# B&R Automation Studio project Nitto (part 11)

#### Bibliothek.fun - Exportierte Funktionen und Funktionsblöcke
```iecst
(********************************************************************
 * COPYRIGHT -- Microsoft
 ********************************************************************
 * Library: Bibliothek
 * Datei: Bibliothek.fun
 * Autor: Awalz
 * Erstellt: 31. März 2014
 ********************************************************************
 * Funktionen und Funktionsblöcke der Library Bibliothek
 ********************************************************************)

FUNCTION_BLOCK FB_CONST_MACHINE_MODES (*TODO: Bitte Kommentar hier einzufügen*)
	VAR_OUTPUT
		MANUAL : INT := 0;
		AUTOMATIC : INT := 1;
		PRODUCTION : INT := 2;
		SAFETYSTOP : INT := 7;
		RESET : INT := 8;
		EMERGENCYSTOP : INT := 9; (*texts : ARRAY[MANUAL..EMERGENCYSTOP] OF STRING[20] := ['MANUAL','AUTOMATIC','PRODUCTION','***3***','***4***','***5***','***6***','SAFETYSTOP','RESET','EMERGENCYSTOP'];*)
		texts : ARRAY[0..9] OF STRING[20] := ['MANUAL','AUTOMATIC','PRODUCTION','***3***','***4***','***5***','***6***','SAFETYSTOP','RESET','EMERGENCYSTOP'];
	END_VAR
END_FUNCTION_BLOCK

FUNCTION_BLOCK FB_CONST_AXIS_ACTIONS (*TODO: Bitte Kommentar hier einzufügen*)
	VAR_OUTPUT
		NOACTION : INT := 0;
		START : INT := 1;
		CALIBR : INT := 2;
		JOG_POS : INT := 3;
		JOG_NEG : INT := 4;
		SETPOS : INT := 6;
		CPLON : INT := 7;
		CPLOFF : INT := 8;
		STOP : INT := 9;
		RESET : INT := 10;
		OPEN : INT := 11; (* Break Open*)
		CLOSE : INT := 12; (* Break Close*)
		WRITE : INT := 13; (* Write Parameter*)
		READ : INT := 14; (* Read Parameter*)
		MOVE_VELOCITY : INT := 15;
		POWER_ON : INT := 16;
		VAXIS_ON : INT := 17;
		POWER_OFF : INT := 18;
		MOVE_CYCLIC_VELOCITY : INT := 20;
		SETPOSREL : INT := 21;
		SETPOSREL_NOLIMIT : INT := 22;
		EMERGENCY_DECELERATION : REAL := 1111111; (*200m/min 200*16666.67/2 in 2 sek*)
		texts : ARRAY[0..19] OF STRING[15] := ['NOACTION','START','CALIBR','JOG_POS','JOG_NEG','SETPOS','SETPOS','CPLON','CPLOFF','STOP','RESET','OPEN','CLOSE','WRITE','READ','MOVE_VELO','POWER_ON','VAXIS_ON','POWER_OFF'];
	END_VAR
END_FUNCTION_BLOCK

FUNCTION_BLOCK FB_CONST_MASCHINE (*TODO: Bitte Kommentar hier einzufügen*)
	VAR_INPUT
		MACHINEMODES : FB_CONST_MACHINE_MODES;
		AXIS : FB_CONST_AXIS_ACTIONS;
		LAMP : FB_CONST_LAMP;
		CUTTINGUNIT : FB_CONST_CUTTINGUNIT;
		UNITMODEs : FB_CONST_UNIT_MODES;
		ALARMS : FB_CONST_ALARMS;
	END_VAR
END_FUNCTION_BLOCK

FUNCTION_BLOCK FB_ClkPulse (*TODO: Bitte Kommentar hier einzufügen*)
	VAR_INPUT
		enable : BOOL;
		TimeOn : TIME := T#100ms;
		TimeOff : TIME := T#100ms;
	END_VAR
	VAR_OUTPUT
		Output : BOOL := FALSE;
	END_VAR
	VAR CONSTANT
		CLOCK_ON : INT := 0;
		CLOCK_WAIT_ON : INT := 1;
		CLOCK_WAIT_OFF : INT := 3;
	END_VAR
	VAR
		state : INT := CLOCK_ON;
		timer : TON;
	END_VAR
END_FUNCTION_BLOCK

FUNCTION_BLOCK FB_Clk (*TODO: Bitte Kommentar hier einzufügen*)
	VAR_OUTPUT
		c500 : FB_ClkPulse := (enable:=TRUE,TimeOn:=T#500ms,TimeOff:=T#500ms);
		c200 : FB_ClkPulse := (enable:=TRUE,TimeOn:=T#200ms,TimeOff:=T#200ms);
		c1000 : FB_ClkPulse := (enable:=TRUE,TimeOn:=T#1000ms,TimeOff:=T#1000ms);
		c5000 : FB_ClkPulse := (enable:=TRUE,TimeOn:=T#5000ms,TimeOff:=T#5000ms);
	END_VAR
END_FUNCTION_BLOCK

FUNCTION_BLOCK FB_CONST_LAMP (*TODO: Bitte Kommentar hier einzufügen*)
	VAR_OUTPUT
		OFF : INT := 0;
		ON : INT := 1;
		BLINK200 : INT := 2;
		BLINK500 : INT := 3;
		BLINK1000 : INT := 4;
		BLINK5000 : INT := 5;
	END_VAR
END_FUNCTION_BLOCK

FUNCTION_BLOCK FB_CONST_CUTTINGUNIT (*TODO: Bitte Kommentar hier einzufügen*)
	VAR_INPUT
		MODEs : FB_CONST_CUTTINGUNIT_MODES;
		CMDs : FB_CONST_CUTTINGUNIT_CMDS;
		ERRORs : FB_CONST_CUTTINGUNIT_ERRORS;
		TOOLs : FB_CONST_CUTTINGUNIT_TOOLS;
	END_VAR
END_FUNCTION_BLOCK

FUNCTION_BLOCK FB_CONST_CUTTINGUNIT_MODES (*TODO: Bitte Kommentar hier einzufügen*)
	VAR_OUTPUT
		DISABLE : UDINT := 0; (*BYTE *) (* nicht gekoppelt zur Achse vom Mastermodul *)
		FREE_RUN : UDINT := 1; (*BYTE *) (* freies Schneiden *)
		SYNC_RUN : UDINT := 2; (*BYTE *) (* synchronisieren z.B. Registermarken *)
		CROSS_CUT : UDINT := 3;
		END_MODE : UDINT := 10; (*BYTE *)
		texts : ARRAY[1..4] OF STRING[20] := ['DISABLE','FREE_RUN','SYNC_RUN','CROSS_CUT'];
	END_VAR
END_FUNCTION_BLOCK

FUNCTION_BLOCK FB_CONST_CUTTINGUNIT_CMDS (*TODO: Bitte Kommentar hier einzufügen*)
	VAR_OUTPUT
		NO_CMD : INT := 0;
		CALIBR : INT := 1;
		INIT : INT := 2;
		CPL_ON : INT := 3;
		CPL_OFF : INT := 4;
		DEINIT : INT := 5;
		SYNC : INT := 6;
		MOVEFW : INT := 7;
		MOVEBW : INT := 8;
		RESET : INT := 9;
		SETDATA : INT := 10;
		ABORT : INT := 11;
		texts : ARRAY[1..11] OF STRING[20] := ['NO_CMD','CALIBR','INT','CPL_ON','CPL_OFF','DEINIT','SYNC','MOVEFW','MOVEBW','RESET','SETDATA','ABORT'];
	END_VAR
END_FUNCTION_BLOCK

FUNCTION_BLOCK FB_CONST_UNIT_MODES (*TODO: Bitte Kommentar hier einzufügen*)
	VAR_OUTPUT
		DISABLE : UDINT := 0; (*BYTE*)
		ENABLE : UDINT := 1; (*BYTE*)
		AXIS_OFF : DINT := 2;
		texts : ARRAY[0..2] OF STRING[20] := ['DISABLE','ENABLE','AXIS_OFF'];
	END_VAR
END_FUNCTION_BLOCK

FUNCTION_BLOCK FB_CUTTINGUNIT_CMD (*TODO: Bitte Kommentar hier einzufügen*)
	VAR_INPUT
		value : INT;
		set : BOOL;
	END_VAR
	VAR_OUTPUT
		text : STRING[20];
	END_VAR
	VAR
		CONST : FB_CONST_MASCHINE;
	END_VAR
END_FUNCTION_BLOCK

FUNCTION_BLOCK FB_TensionMeasure (*TODO: Bitte Kommentar hier einzufügen*)
	VAR_INPUT
		offsetVisu : LREAL;
		data : FB_TENSIONMEASUREDATA;
		init : BOOL;
	END_VAR
	VAR_OUTPUT
		status : FB_ModulStatus;
		actValue : LREAL;
	END_VAR
	VAR
		CyclicWrite : MC_BR_CyclicWrite;
		PIDControler : LCRPID; (* PID REGLER*)
		LCRPIDpara_TM : LCRPIDpara; (* Parameter für PID REGLER*)
		FilterPT1 : LCRPT1e;
		CONST : FB_CONST_MASCHINE;
	END_VAR
	VAR CONSTANT
		STEP_TM_INIT1 : USINT := 0; (*Initialisation step 1*)
		TENSION_T_FILTER : REAL := 0.016; (*tension filter time [s]*)
		STEP_TM_WAIT_POWER_ENABLED : USINT := 7; (*Wait until all available axes are enabled*)
		STEP_TM_READY : USINT := 10; (*General state after initialisation, waining for commands*)
		STEP_TM_LOAD_PARA_START : USINT := 20; (*Start parameter loading (e.g. PID controller parameter)*)
		STEP_TM_WAIT_LOAD_PARA_DONE : USINT := 21; (*Wait for parameter being loaded *)
		STEP_TM_WAIT_SWITCH_CTRL_ON : USINT := 40; (*Switch PID controller on*)
		STEP_TM_CTRL_ACTIVE : USINT := 41; (*Wait for commands in active control*)
		STEP_TM_CTRL_PAUSE : USINT := 42; (*Pausing control until the master velocity is back in the required range*)
		STEP_TM_CTRL_OFF : USINT := 43; (*Switch off web tension control*)
	END_VAR
END_FUNCTION_BLOCK

FUNCTION_BLOCK FB_TENSIONMEASUREDATA (*TODO: Bitte Kommentar hier einzufügen*)
	VAR_INPUT
		mode : UDINT; (*BYTE;*)
		setvalue : REAL;
	END_VAR
	VAR_OUTPUT
		newRecipe : BOOL;
	END_VAR
END_FUNCTION_BLOCK

FUNCTION_BLOCK FB_Safety (*TODO: Bitte Kommentar hier einzufügen*)
	VAR_INPUT
		ResetSafeMC : BOOL; (*Reset input of SafeMC Function Blocks*)
		ResetStartupInhibit : BOOL; (*Reset emergency functions (quit startup inhibit)*)
		ResetUserSafeMC : BOOL;
		SLSmasterVeloScaled : REAL;
		Control_OFF : BOOL;
		CtrlPowerEmcyDel : BOOL;
		CtrlPowerEmcyUndel : BOOL; (* schaltet die Schützte für 24V Versorgung*)
		EnabDrives : BOOL;
		manuelmode : BOOL;
	END_VAR
	VAR_OUTPUT
		RequestSTO : BOOL; (*Emergency Stop is requested (active low)*)
		RequestSLS : BOOL; (*Safe Limited Speed requested by opening safety doors (active low)*)
		Request_ONdelay : BOOL;
		valid : BOOL;
	END_VAR
END_FUNCTION_BLOCK

FUNCTION_BLOCK FB_ModulStatus (*TODO: Bitte Kommentar hier einzufügen*)
	VAR_INPUT
		id : UINT;
		name : STRING[30];
		isCoupled : BOOL;
		mode : UDINT; (* BYTE;*)
		ready : BOOL;
		reverse : BOOL;
		axiserror : BOOL;
	END_VAR
	VAR_OUTPUT
		modeName : STRING[80];
		error : BOOL;
		AxisState_status : STRING[20];
	END_VAR
	VAR_IN_OUT
		axisState : MC_ReadStatus;
	END_VAR
END_FUNCTION_BLOCK

FUNCTION_BLOCK FB_Ampel (*TODO: Bitte Kommentar hier einzufügen*)
	VAR_INPUT
		Rot : FB_Lamp; (*DiDo_Type;*)
		Gelb : FB_Lamp; (*DiDo_Type;*)
		Gruen : FB_Lamp; (* DiDo_Type;*)
		horn : BOOL;
		hornoff : BOOL;
		hornPuls : FB_Lamp;
		ondelay : TIME;
	END_VAR
	VAR_OUTPUT
		horn_o : BOOL;
	END_VAR
	VAR_IN_OUT
		clk : FB_Clk;
	END_VAR
	VAR
		rtrig : R_TRIG;
		timer_TOF : TOF;
		timer_TON : TON;
	END_VAR
END_FUNCTION_BLOCK

FUNCTION_BLOCK FB_Lamp (*TODO: Bitte Kommentar hier einzufügen*)
	VAR_INPUT
		aktion : INT := 0;
	END_VAR
	VAR_OUTPUT
		led : BOOL := FALSE;
		ledinv : BOOL := FALSE;
		button : BOOL;
		rtrig : R_TRIG;
		ftrig : F_TRIG;
	END_VAR
	VAR_IN_OUT
		clk : FB_Clk;
	END_VAR
	VAR
		CONST : FB_CONST_MASCHINE;
		output : BOOL := FALSE;
	END_VAR
END_FUNCTION_BLOCK

FUNCTION_BLOCK FB_KeyLamp (*TODO: Bitte Kommentar hier einzufügen*)
	VAR_INPUT
		LDT : FB_Lamp;
	END_VAR
	VAR_IN_OUT
		clk : FB_Clk;
	END_VAR
END_FUNCTION_BLOCK

FUNCTION_BLOCK FB_UnitChkStatus (*TODO: Bitte Kommentar hier einzufügen*)
	VAR_INPUT
		enable : BOOL;
		setMode : UDINT; (*BYTE;*)
	END_VAR
	VAR_OUTPUT
		ready : BOOL;
	END_VAR
	VAR_IN_OUT
		status : FB_ModulStatus;
	END_VAR
	VAR
		CONST : FB_CONST_MASCHINE;
	END_VAR
END_FUNCTION_BLOCK

FUNCTION_BLOCK FB_PullBreakClampToggle (*TODO: Bitte Kommentar hier einzufügen*)
	VAR_INPUT
		buttomToggle : FB_KeyLamp;
		buttomToggle2 : FB_KeyLamp;
		limiterSwitchDrvSide : BOOL;
		limiterSwitchOpSide : BOOL;
		isup : BOOL;
		isdown : BOOL;
		enable : BOOL;
		init : BOOL;
		onewayini : BOOL;
	END_VAR
	VAR_OUTPUT
		toUp_o : BOOL;
		toDown_o : BOOL;
		limiterBackward_o : BOOL;
		limiterForward_o : BOOL;
	END_VAR
	VAR_IN_OUT
		clk : FB_Clk;
	END_VAR
	VAR
		Time1 : TON;
		state : USINT := 0;
		CONST : FB_CONST_MASCHINE;
	END_VAR
END_FUNCTION_BLOCK

FUNCTION_BLOCK FB_ErrorHdl (*TODO: Bitte Kommentar hier einzufügen*)
	VAR_INPUT
		set : BOOL;
		reset : BOOL;
		flag : BOOL;
		id : DINT;
		state : DINT;
		text : STRING[256];
		fnc : STRING[128];
	END_VAR
END_FUNCTION_BLOCK

FUNCTION_BLOCK FB_Panel (*TODO: Bitte Kommentar hier einzufügen*)
	VAR_INPUT
		Emergency : FB_KeyLamp;
		EMCY_Button : BOOL;
		LDTRESET : FB_KeyLamp;
		LDTStop : FB_KeyLamp;
		LDTAutomatic : FB_KeyLamp;
		LDTJOG : FB_KeyLamp;
		LDTControlON : FB_KeyLamp;
		LDTControlOFF : FB_KeyLamp;
	END_VAR
	VAR_OUTPUT
		clk : FB_Clk;
		EMCY_Button_o : INT;
	END_VAR
END_FUNCTION_BLOCK

FUNCTION_BLOCK FB_CONVEYOR_DATA (*TODO: Bitte Kommentar hier einzufügen*)
	VAR_INPUT
		gap : LREAL;
		pcs : INT;
		newParam2 : BOOL;
	END_VAR
END_FUNCTION_BLOCK

FUNCTION_BLOCK FB_MASTERMODUL_DATA (*TODO: Bitte Kommentar hier einzufügen*)
	VAR_INPUT
		speedToCycleWebturrit : REAL;
		startSpeed : REAL;
		maxSpeed : REAL;
		periodLength : REAL;
		lenght1 : REAL;
		lenght2 : REAL;
	END_VAR
END_FUNCTION_BLOCK

FUNCTION_BLOCK FB_MessageInstance (*TODO: Bitte Kommentar hier einzufügen*)
	VAR_INPUT
		active : BOOL;
		InstanceId : UDINT; (* Aggregat, Instaziertes Objekt *)
		ErrorId : UDINT;
		StationName : STRING[20];
	END_VAR
	VAR_OUTPUT
		err : FB_ErrorHdl;
		busy : BOOL;
	END_VAR
	VAR
		state : INT;
		sFormatString : STRING[29] := '';
		arrParaPointer : ARRAY[1..3] OF DINT;
		sPara1 : STRING[20];
		nPara2 : DINT;
		nPara3 : DINT; (*fbLogEvent:		ADSLOGEVENT := ( PORT:=110,
											  TMOUT := T#2s,
											  EventConfigData := ( 	Class := TCEVENTCLASS_ALARM,
																			Prio := TCEVENTPRIO_IMPLICIT,
																			ProgId := 'TcEventFormatter.TcXmlFormatter',
																			StreamType := TCEVENTSTREAM_NORMAL,
																			bQuitRequired := FALSE
																		)
											);*)
	END_VAR
END_FUNCTION_BLOCK

FUNCTION_BLOCK FB_WinderData (*TODO: Bitte Kommentar hier einzufügen*)
	VAR_INPUT
		recipeData : FB_WinderRecipeData;
		machData : FB_WinderMachData;
	END_VAR
END_FUNCTION_BLOCK

FUNCTION_BLOCK FB_WinderRecipeData (*TODO: Bitte Kommentar hier einzufügen*)
	VAR_INPUT
		stopDiam : UDINT;
		warnDiam : UDINT;
		minDiamTension : UDINT; (*Mode*)
		maxDiamTension : UDINT; (*Mode*)
		mode : UDINT; (*Mode*)
		reverse : BOOL;
		dancersolPos : REAL;
	END_VAR
END_FUNCTION_BLOCK

FUNCTION_BLOCK FB_WinderMachData (*TODO: Bitte Kommentar hier einzufügen*)
	VAR_INPUT
		coreDiam : UDINT;
		frictionCompensation : USINT := 0;
		velocityOverride : USINT := 0;
		GEAR_RATIO : REAL;
		axistyp : SINT; (* (-1: winder, +1: unwinder).*)
	END_VAR
END_FUNCTION_BLOCK

FUNCTION_BLOCK FB_ScalingPerimeter (*TODO: Bitte Kommentar hier einzufügen*)
	VAR_INPUT
		realperimeter : REAL; (* Umfang des Wekrzeuges *)
		NumberToolSegments : USINT; (*Anzahl der Nutzen auf dem Werkzeug/Stanzblech*)
	END_VAR
	VAR_OUTPUT
		Scaledperimeter : UDINT;
		ToolSegmentPeriod : UDINT;
	END_VAR
	VAR
		Remainder : DINT;
	END_VAR
END_FUNCTION_BLOCK

FUNCTION_BLOCK FB_CUTTINGUNIT_STATUS (*TODO: Bitte Kommentar hier einzufügen*)
	VAR_INPUT
		id : UINT;
		tableid : UINT;
		name : STRING[30];
		dataOk : BOOL;
		isCalibrated : BOOL;
		isInitialized : BOOL;
		isCoupled : BOOL;
		isSynchronized : BOOL; (*	errors:					FB_CUTTINGUNIT_ERRORS;*) (*tmpData:				FB_CUTTINGUNIT_TMPDATA;*)
		errorstop : BOOL;
		extReady : BOOL := TRUE;
		mode : FB_CUTTING_MODE;
	END_VAR
	VAR_OUTPUT
		ready : BOOL;
		tmpCalibrated : BOOL;
		AxisState_status : STRING[20];
	END_VAR
	VAR_IN_OUT
		recipeMode : UDINT; (*	BYTE;*)
		axisState : MC_ReadStatus;
	END_VAR
	VAR
		CONST : FB_CONST_MASCHINE;
	END_VAR
END_FUNCTION_BLOCK

FUNCTION_BLOCK FB_CUTTING_MODE (*TODO: Bitte Kommentar hier einzufügen*)
	VAR_INPUT
		value : UDINT; (*BYTE;*)
	END_VAR
	VAR_OUTPUT
		text : STRING[20];
	END_VAR
	VAR
		CONST : FB_CONST_MASCHINE;
	END_VAR
END_FUNCTION_BLOCK

FUNCTION_BLOCK FB_PowerBridge (*TODO: Bitte Kommentar hier einzufügen*)
	VAR_INPUT
		bridgedownbutton : FB_CLAMP;
		withpressureSensor : BOOL;
		movebutton : FB_KeyLamp;
	END_VAR
	VAR_OUTPUT
		pressuredrvside : INT;
		pressureOperside : INT;
		button : BOOL; (*Button in der Visu*)
		valveOut : BOOL;
		pressurepresent : BOOL;
		toggle : FB_PullBreakClampToggle;
	END_VAR
	VAR_IN_OUT
		clk : FB_Clk;
	END_VAR
	VAR
		KNpressuredrvside : REAL;
		KNpressureOperside : REAL;
		pressurereference : REAL;
	END_VAR
	VAR CONSTANT
		SCALE_10V_TO_KN : REAL := (10.0/32767.0); (*10.0 V = 10 kN; 10.0 V = 32767*)
	END_VAR
END_FUNCTION_BLOCK

FUNCTION_BLOCK FB_CONST_CUTTINGUNIT_ERRORS (*TODO: Bitte Kommentar hier einzufügen*)
	VAR_OUTPUT
		REF_ERROR_UNIT_CLOSED : INT := 1;
		AXISERROR : INT := 2;
		SAFETY_SPEED : INT := 3;
		HAUBE1_VORN_OFFEN : INT := 8;
		HAUBE2_HINTEN_OFFEN : INT := 9;
		RECIPE_MODE_UNDEF : INT := 30;
		RECIPE_TOOLNR : INT := 31;
		RECIPE_SHAPE_CONFIG : INT := 32;
		CUTTER_DIAMETER : INT := 33;
		CUTTER_ZAEHNE : INT := 34;
		ANVILROLLER_ZAEHNE : INT := 35;
		ERROR_TABLE_CALC : INT := 36;
	END_VAR
END_FUNCTION_BLOCK

FUNCTION_BLOCK FB_CONST_CUTTINGUNIT_TOOLS (*TODO: Bitte Kommentar hier einzufügen*)
	VAR_OUTPUT
		MIN_TOOLS : INT := 1;
		MAX_TOOLS : INT := 1000;
	END_VAR
END_FUNCTION_BLOCK

FUNCTION_BLOCK FB_TurnGrWinKeysbox (*TODO: Bitte Kommentar hier einzufügen*)
	VAR_INPUT
		GridWinrightkey : FB_CLAMP;
		GridWinleftkey : FB_CLAMP;
		feederturnkey : FB_KeyLamp;
	END_VAR
	VAR_OUTPUT
		feederlimitswitch : BOOL;
		feederturn : BOOL;
		feederright : BOOL;
	END_VAR
	VAR_IN_OUT
		clk : FB_Clk;
	END_VAR
END_FUNCTION_BLOCK

FUNCTION_BLOCK FB_SPLICETABLE (*TODO: Bitte Kommentar hier einzufügen*)
	VAR_INPUT
		disable : BOOL;
		clampBefore : FB_CLAMP;
		clampAfter : FB_CLAMP;
	END_VAR
	VAR_OUTPUT
		ready : BOOL;
	END_VAR
	VAR_IN_OUT
		clk : FB_Clk;
	END_VAR
END_FUNCTION_BLOCK

FUNCTION_BLOCK FB_CLAMP (*TODO: Bitte Kommentar hier einzufügen*)
	VAR_INPUT
		buttonDown : FB_KeyLamp;
		buttonvisu : BOOL;
		toDown_o : BOOL;
		disable : BOOL;
	END_VAR
	VAR_IN_OUT
		clk : FB_Clk;
	END_VAR
	VAR
		visutrigg : R_TRIG;
		CONST : FB_CONST_MASCHINE;
	END_VAR
END_FUNCTION_BLOCK

FUNCTION_BLOCK FB_Cylinder (*TODO: Bitte Kommentar hier einzufügen*)
	VAR_INPUT
		upVISU : BOOL;
		downVISU : BOOL;
		buttonUP : BOOL;
		buttonDown : BOOL;
		Enable : BOOL;
		up_o : BOOL;
		down_o : BOOL;
	END_VAR
	VAR_OUTPUT
		isUp : BOOL;
		isDown : BOOL;
		isdowndelayed : BOOL;
	END_VAR
	VAR
		timer : TON;
	END_VAR
END_FUNCTION_BLOCK

FUNCTION_BLOCK FB_Hydraulic (*TODO: Bitte Kommentar hier einfügen*) (*$GROUP=Anwender*)
	VAR_INPUT
		enable : BOOL;
		buttonDown : BOOL;
		buttonUp : BOOL;
		limitswitch : BOOL; (* kein Endschalter für untern da nur Ventile aufgemacht werden und der Wickler drucklos bis zum Ende fährt*)
	END_VAR
	VAR_OUTPUT
		go_up : BOOL; (*go_down:		BOOL;*) (* da kein Ventil angesteuert wird nur das Ventil für hoch gelüftet wird*)
		commonValve : BOOL;
		LED_is_up : BOOL;
		LED_is_down : BOOL;
		pumpe : BOOL;
	END_VAR
END_FUNCTION_BLOCK

FUNCTION_BLOCK FB_UnwinderfeederCtrl (*TODO: Bitte Kommentar hier einfügen*) (*$GROUP=Anwender*)
	VAR_INPUT
		cmd : INT;
		buttonRequestOpSide : FB_KeyLamp;
		buttonRightOpSide : FB_KeyLamp;
		buttonLeftOpSide : FB_KeyLamp;
		buttonRequestDrvSide : FB_KeyLamp;
		buttonRightDrvSide : FB_KeyLamp;
		buttonLeftDrvSide : FB_KeyLamp;
		LimitSwitchRight : BOOL;
		LimitSwitchLeft : BOOL;
		axisREF : UDINT;
		UnwFeeder_HW : SdcHwCfg_typ := (0);
		UnwFeeder_DrvIf : SdcDrvIf16_typ := (0);
		UnwFeeder_DiDoIf : SdcDiDoIf_typ := (0);
		UnwFeeder_ModuleOk : BOOL := 0;
		UnwFeederErrorAckn : BOOL;
		BasicControl : basic_typ;
	END_VAR
	VAR_OUTPUT
		feederFUleft : BOOL;
		feederFUright : BOOL;
		brakerelease : BOOL;
		ampelgelb : BOOL;
		horn : BOOL;
		MC_ReadStatus_0 : MC_ReadStatus;
		busy : BOOL;
		status : FB_ModulStatus;
	END_VAR
	VAR_IN_OUT
		machineaxis : FB_AxisCtrl;
		clk : FB_Clk;
	END_VAR
	VAR
		AxisStep : INT;
		cmdtmp : INT;
		trigOPSide : BOOL;
		trigDrvSide : BOOL;
		braketimer : BOOL;
		MC_BR_ReadDriveStatus_0 : MC_BR_ReadDriveStatus;
		firststart : BOOL := TRUE;
		State : USINT;
		CONST : FB_CONST_MASCHINE;
		MC_BR_JogVelocity_0 : MC_BR_JogVelocity;
		pAxis : REFERENCE TO ACP10AXIS_typ;
		MC_Power_0 : MC_Power;
		MC_Stop_0 : MC_Stop;
		MC_Reset_0 : MC_Reset;
		Start_timer : BOOL; (*timer_TOF : TON;*)
		timer_TON : TON;
		timerOPside_TOF : TOF; (*Scahltet den Regler ab und damit fällt die Bremse zu*)
		timerDrvside_TOF : TOF;
		timer_TP : TP;
	END_VAR
	VAR CONSTANT
		STATE_READY : INT := 0;
		STATE_POWER_ON : INT := 10;
		STATE_POWER_OFF : INT := 11;
		STATE_ERROR_RESET : INT := 12;
		STATE_QUIT : INT := 20;
		ST_WAIT : USINT := 0;
		ST_REQUEST : USINT := 10;
		ST_REQUEST_OpSide : USINT := 20;
		ST_REQUEST_DrvSide : USINT := 30;
		ST_END : USINT := 40;
	END_VAR
END_FUNCTION_BLOCK

FUNCTION_BLOCK FB_DUBBLEUUNWINDERDATA (*TODO: Bitte Kommentar hier einfügen*) (*$GROUP=Anwender*)
	VAR_INPUT
		undwinderDRV : FB_WinderData; (*drive side*)
		unwinderOP : FB_WinderData; (*operator side*)
	END_VAR
END_FUNCTION_BLOCK

FUNCTION_BLOCK FB_UNWINDERUNITSTATUS (*TODO: Bitte Kommentar hier einfügen*) (*$GROUP=Anwender*)
	VAR_INPUT
		statusDrv : FB_ModulStatus;
		statusOP : FB_ModulStatus;
	END_VAR
END_FUNCTION_BLOCK

FUNCTION_BLOCK FB_limitswitch (*TODO: Bitte Kommentar hier einfügen*) (*$GROUP=Anwender*)
	VAR_INPUT
		limitSWupper : BOOL;
		limitSWlower : BOOL;
		mechbrake : BOOL;
	END_VAR
END_FUNCTION_BLOCK

FUNCTION_BLOCK FB_StartStopbox (*TODO: Bitte Kommentar hier einfügen*) (*$GROUP=Anwender*)
	VAR_INPUT
		start : FB_KeyLamp;
		stop : FB_KeyLamp;
		jog : FB_KeyLamp;
	END_VAR
	VAR_IN_OUT
		clk : FB_Clk;
	END_VAR
END_FUNCTION_BLOCK

FUNCTION_BLOCK FB_SummeryStarStop (*TODO: Bitte Kommentar hier einfügen*) (*$GROUP=Anwender*)
	VAR_INPUT
		boxunwinder : FB_StartStopbox;
		boxwebbuffer : FB_StartStopbox;
		boxcutting1 : FB_StartStopbox;
		boxlongcutter : FB_StartStopbox;
		boxconveyor : FB_StartStopbox;
	END_VAR
	VAR_OUTPUT
		start : BOOL;
		stop : BOOL;
		jog : BOOL;
	END_VAR
	VAR_IN_OUT
		panel : FB_Panel;
		clk : FB_Clk;
	END_VAR
END_FUNCTION_BLOCK

FUNCTION_BLOCK FB_WebGuiding (*TODO: Bitte Kommentar hier einfügen*) (*$GROUP=Anwender*)
	VAR_INPUT
		enable : BOOL;
		center : BOOL;
		auto : BOOL;
		hand : BOOL;
		moveRight : BOOL;
		moveLeft : BOOL;
		hardwareOK : BOOL;
	END_VAR
	VAR_OUTPUT
		manual : BOOL;
		neutral : BOOL;
		automatic : BOOL;
		centerSelect : BOOL;
		handSelect : BOOL;
		autoSelect : BOOL;
		active : BOOL;
		arrowRight : BOOL;
		arrowLeft : BOOL;
		hardwareActive : BOOL;
	END_VAR
	VAR
		TP_01 : TP;
		Start_timer : BOOL;
		handtrigg : R_TRIG;
		centertrigg : R_TRIG;
		autotrigg : R_TRIG;
	END_VAR
END_FUNCTION_BLOCK

FUNCTION_BLOCK FB_SetGearRatio (*TODO: Bitte Kommentar hier einfügen*) (*$GROUP=Anwender*)
	VAR_INPUT
		UpdateRecipe : BOOL;
		setvalueVisuRecipe : REAL;
		enable : BOOL;
		step1 : BOOL;
		step10 : BOOL;
		step100 : BOOL;
		gearup : BOOL;
		gearlow : BOOL;
		Selectstep1 : BOOL;
		Selectstep10 : BOOL;
		Selectstep100 : BOOL;
		Selectenable : BOOL;
		limitvisupos : REAL;
		limitvisuneg : REAL;
		limitratiopos : INT;
		limitrationeg : INT;
		init : BOOL;
	END_VAR
	VAR_OUTPUT
		trigger : BOOL;
		ratioNumeratorOut : INT;
		ratioDenominator : UINT := 1000;
		setvalueVisu : REAL;
		stepvisu : REAL;
		ratio_inProcent_visu : REAL;
	END_VAR
	VAR
		offsetrecipe : REAL;
		trigP : R_TRIG;
		trigN : R_TRIG;
		ratio : INT := 1000;
		ratiotmp : INT;
		step : INT;
		TP_01 : TP;
		Start_timer : BOOL;
	END_VAR
END_FUNCTION_BLOCK

FUNCTION_BLOCK FB_MarkPoints (*TODO: Bitte Kommentar hier einfügen*) (*$GROUP=Anwender*)
	VAR_INPUT
		MC_BR_TouchProbe_0 : MC_BR_TouchProbe;
		reset : BOOL;
		Enable : BOOL;
		TriggerInput : MC_BR_TRIGGER_REF; (*Input that is used as event source*)
		Axis : UDINT; (*Axis reference of slave*)
		SearchRM : BOOL; (*Initiate search of new RM on positive edge*)
		CutMasterPosition : DINT; (*Uncorrected next cut position [Master Units]*)
		RegMarkPosition : DINT; (*RegMark offset relative to cut position [Master Units]*)
		WindowNegative : REAL; (*Range before the expected position in which the trigger signal may occur [Master Units]*)
		WindowPositive : REAL; (*Range after the expected position in which the trigger signal may occur [Master Units]*)
		ProductLength : REAL; (*Interval between two expected trigger positions [Master Units]*)
		markpointlist : FB_Markpointarray;
	END_VAR
	VAR_OUTPUT
		RecordedValue : DINT; (*Most recent RM position [Master Units]*)
		lastrecocordedValue : DINT; (*last Position befor RM lost [Master Units]*)
		ProbeCounter : UDINT; (*Number of valid trigger events. Reset by "SearchRM"*)
		MissedTriggers : UDINT; (*Number of invalid or missed trigger events. Reset by "SearchRM"*)
		CorrectionValue : DINT; (*Deviation between corrected and uncorrected cut position [Master Units]. Can be used as a relative distance for correction movements.*)
		CorrectionValid : BOOL; (*TRUE for 1 cycle if "CorrectionValue" is valid. Can be used to trigger correction movements.*)
		ActProductLength : REAL; (*Actual measured product length*)
		Active : BOOL; (*FB is enabled - waiting for a trigger event*)
		Busy : BOOL; (*FB is not yet finished*)
		Error : BOOL; (*Error occurred in FB*)
		ErrorID : UINT; (*Error number*)
	END_VAR
END_FUNCTION_BLOCK

FUNCTION_BLOCK FB_CROSSCUTPAR (*TODO: Bitte Kommentar hier einfügen*) (*$GROUP=Anwender*)
	VAR_INPUT
		StartMasterVelocity : REAL; (*Master velocity at very first cut [Master Units/ s]*)
		MaxMasterVelocity : REAL; (*Maximum master velocity [Master Units/ s]*)
		Insetting : REAL; (*Insetting ratio for calculation of CutRangeMaster [%]*)
		MaxCorrection : DINT; (*Maximum correction movement per product cycle [Master Units]*)
		CutStartPos : DINT; (*Start of synchronisation within slave period [Slave Units]*)
		CutEndPos : DINT; (*End of synchronisation within slave period [Slave Units]*)
		CutRangeMaster : REAL;
		CutRangeSlave : REAL;
		ProductLength : REAL;
		CutPosition : REAL;
		StartMode : UINT;
		ProductLengthCorrection : REAL;
		MasterStartDistance : REAL;
		StartInterval : REAL;
		MinCutRangeSlave : REAL; (*Minimum synchronization distance [Slave Units]*)
		MinCompRangeSlave : REAL; (*Minimum effective compensation distance [Slave Units]*)
	END_VAR
END_FUNCTION_BLOCK

FUNCTION_BLOCK FB_GetNextCuttPos (*TODO: Bitte Kommentar hier einfügen*) (*$GROUP=Anwender*)
	VAR_INPUT
		Enable : BOOL;
		reset : BOOL;
		donecut : BOOL; (*wait until Cutter is done with a cut*)
		RecordedValue : DINT; (*Recorded RegMark position, e.g. from a MC_BR_Touchprobe instance [Master Units]*)
		RecordedValueValid : BOOL;
		CutPosition : DINT; (*Uncorrected next cut position [Master Units]*)
		DistanceToSensor : DINT; (*Distance between tool and sensor [Master Units]*)
		RegMarkPosition : DINT; (*RegMark offset relative to cut position [Master Units]*)
		ProductLength : DINT; (*Product length [Master Units]*) (*	Touchpobe: MC_BR_TouchProbe;*)
		setCutOffset : FB_SetCutOffset;
	END_VAR
	VAR_OUTPUT
		PositionError : DINT; (*Difference between corrected and uncorrected cut position [Master Units]*)
		PositionErrorValid : BOOL; (*TRUE for 1 cycle if "PositionError" is within current product cycle*)
		nextsyncpos : DINT; (* Position für die Sunchronisierung der Stanze /Querschneider*)
		newdata : UDINT;
	END_VAR
	VAR_IN_OUT
		markpoints : FB_MarkPoints;
		scalePerimeter : FB_ScalingPerimeter;
		machinemaster : FB_AxisCtrl;
	END_VAR
	VAR
		masterposMod : DINT;
		IncompensatinRtrig : R_TRIG;
		IncompensatinFtrig : F_TRIG;
		oldCutPosition : DINT;
		tmpCutPosition : DINT;
		actCutPosition : DINT;
		markposMod : DINT;
		ModDistanceToSensor : DINT;
		probecounter : UDINT;
		indx : UDINT;
		counter : UDINT;
		donecounter : UDINT;
		actmarkpos : UDINT;
		State : INT;
		CorrectedCutPosition : DINT;
		PositionErrorTemp : DINT;
	END_VAR
	VAR CONSTANT
		ST_IDLE : INT := 0;
		ST_READ_POS : INT := 1;
		ST_READ_POS_DONE : INT := 2;
	END_VAR
END_FUNCTION_BLOCK

FUNCTION_BLOCK FB_SafeInputs (*TODO: Bitte Kommentar hier einfügen*) (*$GROUP=Anwender*)
	VAR_INPUT
		EMCY_Button1 : BOOL;
		EMCY_Button2 : BOOL;
		EMCY_Button3 : BOOL;
		EMCY_Button4 : BOOL;
		EMCY_Door1 : BOOL;
		EMCY_Door2 : BOOL;
		EMCY_Door3 : BOOL;
		EMCY_Door4 : BOOL;
		EMCY_Door5 : BOOL;
		EMCY_Door6 : BOOL;
		EMCY_pullwireOPs : BOOL;
		EMCY_pullwireDVRs : BOOL;
		EMCY_DoorsClosed : BOOL;
	END_VAR
	VAR_OUTPUT
		EMCY_Button1_o : INT;
		EMCY_Button2_o : INT;
		EMCY_Button3_o : INT;
		EMCY_Button4_o : INT;
		EMCY_Door1_o : INT;
		EMCY_Door2_o : INT;
		EMCY_Door3_o : INT;
		EMCY_Door4_o : INT;
		EMCY_Door5_o : INT;
		EMCY_Door6_o : INT;
		EMCY_pullwireOPs_o : INT;
		EMCY_pullwireDVRs_o : INT;
	END_VAR
END_FUNCTION_BLOCK

FUNCTION_BLOCK FB_Markpointarray (*TODO: Bitte Kommentar hier einfügen*) (*$GROUP=Anwender*)
	VAR_INPUT
		rdpos : DINT; (*read position*)
		offset_posIdent : USINT;
		new_Ident : BOOL;
		reset : BOOL;
	END_VAR
	VAR_OUTPUT
		lastpos : DINT;
		actlenght : DINT;
		actpos : DINT;
		index_out : UDINT;
		valid : BOOL;
	END_VAR
	VAR
		poslist : ARRAY[0..200] OF DINT;
		points : ARRAY[0..200] OF FB_Points;
		in_posIdent : USINT;
		out_posIdent : USINT; (*	out_lastIdent:USINT;*)
		out_actIdent : USINT;
		maxposIdent : USINT;
		bufferRtrig : R_TRIG;
		visuIndex : USINT;
	END_VAR
	VAR CONSTANT
		maxVisuIndex : USINT := 17; (*Größe des angezeigten Registermarkenfeldes in der Visu *)
	END_VAR
END_FUNCTION_BLOCK

FUNCTION_BLOCK FB_SwitchCabinet (*TODO: Bitte Kommentar hier einfügen*) (*$GROUP=Anwender*)
	VAR_INPUT
		EMCY_Buttons : FB_SafeInputs;
		fusePlug1 : BOOL;
		fusePlug2 : BOOL;
		fusePlugCEE : BOOL;
		aircond : BOOL;
		fuseWebGuide1 : BOOL;
		fuseWebGuide2 : BOOL;
	END_VAR
END_FUNCTION_BLOCK

FUNCTION_BLOCK FB_AxisCrtl_Home (*TODO: Bitte Kommentar hier einfügen*) (*$GROUP=Anwender*)
	VAR_INPUT
		cmd : INT;
		position : REAL;
		velocity : REAL;
		override : REAL;
		verzoegerung : REAL;
		ruck : REAL;
		AxisREF : UDINT;
		BasicControl : basic_typ;
		MC_refSwitchConfig_0 : MC_BR_SetHardwareInputs;
	END_VAR
	VAR_OUTPUT
		busy : BOOL;
		MC_BR_ReadDriveStatus_0 : MC_BR_ReadDriveStatus;
		MC_ReadStatus_0 : MC_ReadStatus;
		err : FB_ErrorHdl;
		MC_ReadActualPosition_0 : MC_ReadActualPosition;
	END_VAR
	VAR CONSTANT
		STATE_WAIT : USINT := 0; (*NOACTION*)
		STATE_POWER_ON : USINT := 1; (*START*)
		STATE_HOME : USINT := 2; (*CALIBR*)
		STATE_JOG_POSITIVE : USINT := 3;
		STATE_JOG_NEGATIVE : USINT := 4;
		STATE_IDLE : USINT := 5;
		STATE_STOP : USINT := 9;
		STATE_READY : USINT := 10;
		STATE_HALT : USINT := 12;
		STATE_MOVE_ABSOLUTE : USINT := 13;
		STATE_SETPOS : USINT := 14;
		STATE_MOVE_VELOCITY : USINT := 15;
		STATE_MOVE_ADDITIVE : USINT := 16;
		STATE_VAXIS_ON : USINT := 17;
		STATE_POWER_OFF : USINT := 18;
		STATE_QUIT : USINT := 19;
		STATE_ERROR_AXIS : USINT := 100;
		STATE_ERROR : USINT := 101;
		STATE_ERROR_RESET : USINT := 102;
	END_VAR
	VAR
		MC_Home_0 : MC_Home;
		MC_MoveAbsolute_0 : MC_MoveAbsolute;
		MC_MoveAdditive_0 : MC_MoveAdditive;
		MC_MoveVelocity_0 : MC_MoveVelocity;
		MC_Power_0 : MC_Power;
		MC_ReadActualVelocity_0 : MC_ReadActualVelocity;
		MC_ReadAxisError_0 : MC_ReadAxisError;
		MC_Reset_0 : MC_Reset;
		MC_Stop_0 : MC_Stop;
		MC_Halt_0 : MC_Halt; (*MC_GearIn_0 : MC_GearIn;*)
		AxisStep : UINT := STATE_WAIT;
		CONST : FB_CONST_MASCHINE;
		cmdtmp : INT;
		merker : BOOL;
	END_VAR
END_FUNCTION_BLOCK

FUNCTION_BLOCK FB_AxisCtrl (*TODO: Bitte Kommentar hier einfügen*) (*$GROUP=Anwender*)
	VAR_INPUT
		cmd : INT;
		position : REAL;
		velocity : REAL;
		override : REAL;
		verzoegerung : REAL;
		ruck : REAL;
		AxisREF : UDINT;
		BasicControl : basic_typ;
	END_VAR
	VAR_OUTPUT
		busy : BOOL;
		MC_BR_ReadDriveStatus_0 : MC_BR_ReadDriveStatus;
		MC_ReadStatus_0 : MC_ReadStatus;
		err : FB_ErrorHdl;
		MC_ReadActualPosition_0 : MC_ReadActualPosition;
		MC_ReadActualVelocity_0 : MC_ReadActualVelocity;
	END_VAR
	VAR CONSTANT
		STATE_WAIT : USINT := 0; (*NOACTION*)
		STATE_POWER_ON : USINT := 1; (*START*)
		STATE_HOME : USINT := 2; (*CALIBR*)
		STATE_JOG_POSITIVE : USINT := 3;
		STATE_JOG_NEGATIVE : USINT := 4;
		STATE_IDLE : USINT := 5;
		STATE_STOP : USINT := 9;
		STATE_READY : USINT := 10;
		STATE_HALT : USINT := 12;
		STATE_MOVE_ABSOLUTE : USINT := 13;
		STATE_SETPOS : USINT := 14;
		STATE_MOVE_VELOCITY : USINT := 15;
		STATE_MOVE_ADDITIVE : USINT := 16;
		STATE_VAXIS_ON : USINT := 17;
		STATE_POWER_OFF : USINT := 18;
		STATE_QUIT : USINT := 19;
		STATE_ERROR_AXIS : USINT := 100;
		STATE_ERROR : USINT := 101;
		STATE_ERROR_RESET : USINT := 102;
	END_VAR
	VAR
		MC_Home_0 : MC_Home;
		MC_MoveAbsolute_0 : MC_MoveAbsolute;
		MC_MoveAdditive_0 : MC_MoveAdditive;
		MC_MoveVelocity_0 : MC_MoveVelocity;
		MC_Power_0 : MC_Power;
		MC_ReadAxisError_0 : MC_ReadAxisError;
		MC_Reset_0 : MC_Reset;
		MC_Stop_0 : MC_Stop;
		MC_Halt_0 : MC_Halt; (*MC_GearIn_0 : MC_GearIn;*)
		AxisStep : UINT := STATE_WAIT;
		CONST : FB_CONST_MASCHINE;
		cmdtmp : INT;
		merker : BOOL;
	END_VAR
END_FUNCTION_BLOCK

FUNCTION_BLOCK FB_AxisCtrl_GridFeeder (*TODO: Bitte Kommentar hier einfügen*) (*$GROUP=Anwender*)
	VAR_INPUT
		cmd : INT;
		position : REAL;
		velocity : REAL;
		override : REAL;
		verzoegerung : REAL;
		ruck : REAL;
		AxisREF : UDINT;
		BasicControl : basic_typ;
	END_VAR
	VAR_OUTPUT
		busy : BOOL;
		MC_BR_ReadDriveStatus_0 : MC_BR_ReadDriveStatus;
		MC_ReadStatus_0 : MC_ReadStatus;
		err : FB_ErrorHdl;
		MC_ReadActualPosition_0 : MC_ReadActualPosition;
		MC_ReadActualVelocity_0 : MC_ReadActualVelocity;
	END_VAR
	VAR CONSTANT
		STATE_WAIT : USINT := 0; (*NOACTION*)
		STATE_POWER_ON : USINT := 1; (*START*)
		STATE_HOME : USINT := 2; (*CALIBR*)
		STATE_JOG_POSITIVE : USINT := 3;
		STATE_JOG_NEGATIVE : USINT := 4;
		STATE_IDLE : USINT := 5;
		STATE_STOP : USINT := 9;
		STATE_READY : USINT := 10;
		STATE_HALT : USINT := 12;
		STATE_MOVE_ABSOLUTE : USINT := 13;
		STATE_SETPOS : USINT := 14;
		STATE_MOVE_VELOCITY : USINT := 15;
		STATE_MOVE_ADDITIVE : USINT := 16;
		STATE_VAXIS_ON : USINT := 17;
		STATE_POWER_OFF : USINT := 18;
		STATE_QUIT : USINT := 19;
		STATE_ERROR_AXIS : USINT := 100;
		STATE_ERROR : USINT := 101;
		STATE_ERROR_RESET : USINT := 102;
	END_VAR
	VAR
		MC_Home_0 : MC_Home;
		MC_MoveAbsolute_0 : MC_MoveAbsolute;
		MC_MoveAdditive_0 : MC_MoveAdditive;
		MC_MoveVelocity_0 : MC_MoveVelocity;
		MC_Power_0 : MC_Power;
		MC_ReadAxisError_0 : MC_ReadAxisError;
		MC_Reset_0 : MC_Reset;
		MC_Stop_0 : MC_Stop;
		MC_Halt_0 : MC_Halt; (*MC_GearIn_0 : MC_GearIn;*)
		AxisStep : UINT := STATE_WAIT;
		CONST : FB_CONST_MASCHINE;
		cmdtmp : INT;
		merker : BOOL;
	END_VAR
END_FUNCTION_BLOCK

FUNCTION_BLOCK FB_SetCutOffset (*TODO: Bitte Kommentar hier einfügen*) (*$GROUP=Anwender*)
	VAR_INPUT
		UpdateRecipe : BOOL;
		setvalueVisuRecipe : REAL;
		enable : BOOL;
		maxcorrection : REAL;
		step01 : BOOL;
		step1 : BOOL;
		step10 : BOOL;
		gearup : BOOL;
		gearlow : BOOL;
		Selectstep01 : BOOL;
		Selectstep1 : BOOL;
		Selectstep10 : BOOL;
		Selectenable : BOOL;
		limitvisupos : REAL;
		limitvisuneg : REAL;
	END_VAR
	VAR_OUTPUT
		setvalueVisu : REAL;
		setOffset_o : DINT := 0;
		stepvisu : REAL;
	END_VAR
	VAR
		trigP : R_TRIG;
		trigN : R_TRIG;
		ratio : REAL := 0.0;
		ratiotmp : REAL;
		step : REAL;
		TP_01 : TP;
		Start_timer : BOOL;
	END_VAR
END_FUNCTION_BLOCK

FUNCTION_BLOCK FB_Points (*TODO: Bitte Kommentar hier einfügen*) (*$GROUP=Anwender*)
	VAR_INPUT
		pos : DINT;
		lenght : DINT;
		indx : DINT;
	END_VAR
END_FUNCTION_BLOCK

FUNCTION_BLOCK FB_HandWheel (*TODO: Bitte Kommentar hier einfügen*) (*$GROUP=Anwender*)
	VAR_INPUT
		counterHandWheel : INT;
		limitspeed : REAL;
		actualVelocity : REAL;
		reset : BOOL;
		safetyspeedrequest : BOOL;
	END_VAR
	VAR_OUTPUT
		setVelocity : REAL;
	END_VAR
	VAR
		lastCounterValue : INT;
	END_VAR
	VAR CONSTANT
		velocityStep : REAL := 1666.67; (*0,1m Schritt*)
	END_VAR
END_FUNCTION_BLOCK

FUNCTION_BLOCK FB_Counter (*TODO: Bitte Kommentar hier einfügen*) (*$GROUP=Anwender*)
	VAR_INPUT
		triggerInput : BOOL;
		setPieces : UINT;
		reset : BOOL;
		countPlusVisu : BOOL;
		countMinusVisu : BOOL;
	END_VAR
	VAR_OUTPUT
		counter : UINT;
		counterTemp : UINT;
	END_VAR
	VAR
		R_trig : R_TRIG;
	END_VAR
END_FUNCTION_BLOCK

FUNCTION_BLOCK FB_Counters (*TODO: Bitte Kommentar hier einfügen*) (*$GROUP=Anwender*)
	VAR_INPUT
		counter1 : FB_Counter;
		counter2 : FB_Counter;
		counter3 : FB_Counter;
		counter4 : FB_Counter;
		counter5 : FB_Counter;
		counter6 : FB_Counter;
		counter7 : FB_Counter;
		counter8 : FB_Counter;
		counter9 : FB_Counter;
		setPieces : UINT;
		reset : BOOL;
		visureset : BOOL;
		validpieces : UINT;
		manualButton : BOOL;
		manual : BOOL;
VisuOKButton : BOOL;
	END_VAR
	VAR_OUTPUT
		valid : BOOL;
		Nitto_Table_Full : BOOL;
RedLampOut : BOOL;
GreenLampOut : BOOL;
	END_VAR
	VAR
	zzEdge00000 : BOOL;
	zzEdge00001 : BOOL;
zzEdge00002 : BOOL;
TON_reset : TON;
TON_Nitto_Table_Full : TON;
TP_GreenLampOut : TP;
zzEdge00003 : BOOL;
	END_VAR
END_FUNCTION_BLOCK

FUNCTION_BLOCK FB_Alarms (*TODO: Bitte Kommentar hier einfügen*) (*$GROUP=Anwender*)
	VAR_INPUT
		reset : BOOL;
		alarmlist : ARRAY[0..100] OF BOOL;
	END_VAR
	VAR_OUTPUT
		stopRequest : BOOL;
	END_VAR
	VAR
		i : USINT;
	END_VAR
END_FUNCTION_BLOCK

FUNCTION_BLOCK FB_CONST_ALARMS (*TODO: Bitte Kommentar hier einfügen*) (*$GROUP=Anwender*)
	VAR_OUTPUT
		EMCY_BUTTON_UNWINDER_OP_SIDE : INT := 1;
		EMCY_BUTTON_UNWINDER_DRV_SIDE : INT := 2;
		EMCY_BUTTON_BST : INT := 3;
		EMCY_BUTTON_GRIDWINDER : INT := 4;
		EMCY_BUTTON_PANEL : INT := 5;
		EMCY_BUTTON_LONGCUT_OP_SIDE : INT := 6;
		EMCY_BUTTON_LONGCUT_DRV_SIDE : INT := 7;
		EMCY_BUTTON_CONVEYOR_OP_SIDE : INT := 8;
		EMCY_BUTTON_CONVEYOR_DRV_SIDE : INT := 9;
		EMCY_BUTTON_SCHWITCHCABINET : INT := 10;
		EMCY_OUTSIDE_EXTRUDER : INT := 11;
		EMCY_BUTTON_OUTPUT : INT := 12;
		EMCY_PULLWIRE_OP_SIDE : INT := 15;
		EMCY_PULLWIRE_DRV_SIDE : INT := 16;
		EMCY_DOOR_WEBBUFFER_OP_SIDE : INT := 20;
		EMCY_DOOR_WEBBUFFER_DRV_SIDE : INT := 21;
		EMCY_FRDOOR_WEBBUF_OP_SIDE_LEFT : INT := 22;
		EMCY_FRDOOR_WEBBUF_OP_SIDE_MIDD : INT := 23;
		EMCY_FRDOOR_WEBBUF_OP_SIDE_RIGHT : INT := 24;
		EMCY_FRDOOR_WEBBUF_DRV_SIDE : INT := 25;
		EMCY_DOOR_PBS1 : INT := 26;
		EMCY_DOOR_CUT1_INFEED : INT := 27;
		EMCY_DOOR_CUT1_OUTFEED : INT := 28;
		EMCY_DOOR_LONGCUT : INT := 29;
		EMCY_DOOR_CUT2_INFEED : INT := 30;
		EMCY_DOOR_CUT2_OUTFEED : INT := 31;
		SAFETY_ERROR : INT := 35;
		SAFETY_SPEED : INT := 36;
		MASTER_NOTREADY : INT := 37;
		FUSE_PLUG1 : INT := 40;
		FUSE_PLUG2 : INT := 41;
		FUSE_CEE_PLUG : INT := 42;
		FUSE_WEB_GUIDE_CONTROL_1 : INT := 43;
		WEB_GUIDE_CONTROL_OK_1 : INT := 44;
		FUSE_WEB_GUIDE_CONTROL_2 : INT := 45;
		WEB_GUIDE_CONTROL_OK_2 : INT := 46;
		FUSE_AIR_CONDITIONING : INT := 47;
		AIR : INT := 48;
		UNWINDER_OP_SIDE_DIAMETER_WARN : INT := 50;
		UNWINDER_OP_SIDE_DIAMETER_STOP : INT := 51;
		UNWINDER_OP_SIDE_CLAMP : INT := 52;
		UNWINDER_DRV_SIDE_DIAMETER_WARN : INT := 55;
		UNWINDER_DRV_SIDE_DIAMETER_STOP : INT := 56;
		UNWINDER_DRV_SIDE_CLAMP : INT := 57;
		WEBBUFFER_CLAMP_INFEED : INT := 60;
		WEBBUFFER_EMPTY : INT := 61;
		WEBBUFFER_NOT_REFERENCED : INT := 62;
		SPLICE_TABLE_CLAMP_INFEED : INT := 65;
		SPLICE_TABLE_CLAMP_OUTFEED : INT := 66;
		CUT1_DRIVE_SAFETY : INT := 70;
		CUT1_NOT_REFERENCED : INT := 71;
		GRID_TURN_FEEDER_DRIVE_SAFETY : INT := 75;
		GRID_WINDDER_LEFT_DIAMETER_WARN : INT := 76;
		GRID_WINDDER_LEFT_DIAMETER_STOP : INT := 77;
		GRID_WINDDER_RIGHT_DIAMETER_WARN : INT := 78;
		GRID_WINDDER_RIGHT_DIAMETER_STOP : INT := 79;
		GRID_TURN_FEEDER_NOT_REFERENCED : INT := 80;
		LONGCUT_CLAMP : INT := 85;
		LONGCUT_DRIVE_SAFETY : INT := 86;
		LONGCUT_AXISERRORSTOP : INT := 87;
		LONGCUT_NOT_COUPLED : INT := 88;
		CUT2_DRIVE_SAFETY : INT := 90;
		CUT2_NOT_REFERENCED : INT := 91;
		RECIPEDATA_NOT_LOADED : INT := 95;
		RECIPEDATA_REQUEST_TIMEOUT : INT := 96;
		RECIPEDATA_ERROR : INT := 97;
		PULLBELT_IS_NOT_BELOW : INT := 99;
		CATCHBELT_NOT_COUPLED : INT := 100;
		CONVEYOR_NOT_COUPLED : INT := 101;
	END_VAR
END_FUNCTION_BLOCK

FUNCTION_BLOCK FB_KeysWebbuffer (*TODO: Bitte Kommentar hier einfügen*) (*$GROUP=Anwender*)
	VAR_INPUT
		up : FB_KeyLamp;
		down : FB_KeyLamp;
		home : FB_KeyLamp;
	END_VAR
	VAR_IN_OUT
		clk : FB_Clk;
	END_VAR
END_FUNCTION_BLOCK

FUNCTION_BLOCK FB_MachineSpeed (*TODO: Bitte Kommentar hier einfügen*) (*$GROUP=Anwender*)
	VAR_INPUT
		dancepos : INT;
		setDancerpos : REAL;
		ConveyerVelocity : INT; (*Geschw des HAuptbandes vom Extruders*)
		limitspeed : REAL; (*Limit für den Offset der tatsächlichen Geschw.*)
		reset : BOOL;
		maxMainVelocity : REAL; (*maximale Geschw. der Wert hängt von der Geschw. des Transportbandes bzw. des Extruders Einheit m/min*)
	END_VAR
	VAR_OUTPUT
		setVelocity : REAL;
	END_VAR
	VAR
		rDancepos : REAL;
		velocityramp : LCRRamp;
		TP_01 : TP;
		rtrig : R_TRIG;
		Start_timer : BOOL;
		lowPass : LCRPT1;
		lowPassSpeed : LCRPT1;
		test : INT;
		velocityOffset : REAL;
		inc_to_volt : REAL;
		volt_to_speed : REAL;
		tempvalue : REAL;
	END_VAR
	VAR CONSTANT
		velocityStep : REAL := 166.67; (*0,01m Schritt*)
		highlimitDancerpos : REAL := 400; (*oberste POsition*)
		lowlimitDancerpos : REAL := 830; (*unterste Position des Tänzers*)
		SCALE_INC_TO_V : REAL := (10.0/32767.0); (*(1000.0/32767.0); (*10.0 V = 1000 mm; 10.0 V = 32767*)
		SCALE_10V_TO_MM : REAL := (1000.0/32767.0);
	END_VAR
END_FUNCTION_BLOCK

FUNCTION_BLOCK FB_AxisState (*TODO: Bitte Kommentar hier einfügen*) (*$GROUP=Anwender*)
	VAR_INPUT
		newParam : BOOL;
	END_VAR
	VAR_IN_OUT
		readstatus : MC_ReadStatus;
	END_VAR
	VAR
		stati : ARRAY[0..10] OF BOOL;
		CONST : FB_CONST_AXIS_STATE;
	END_VAR
END_FUNCTION_BLOCK

FUNCTION_BLOCK FB_CONST_AXIS_STATE (*TODO: Bitte Kommentar hier einfügen*) (*$GROUP=Anwender*)
	VAR_OUTPUT
		Error : INT := 1;
		Errorstop : INT := 2;
		Disabled : INT := 3;
		Stopping : INT := 4;
		StandStill : INT := 5;
		DiscreteMotion : INT := 6;
		ContinuousMotion : INT := 7;
		SynchronizedMotion : INT := 8;
		Homing : INT := 9;
		texts : ARRAY[1..9] OF STRING[20] := ['Error','Errorstop','Disabled','Stopping','StandStill','DiscreteMotion','ContinuousMotion','SynchronizedMotion','Homing'];
	END_VAR
END_FUNCTION_BLOCK

FUNCTION_BLOCK FB_SprayCtrl (*TODO: Bitte Kommentar hier einfügen*) (*$GROUP=Anwender*)
	VAR_INPUT
		valveout : BOOL;
		length1 : REAL;
		length2 : REAL;
	END_VAR
	VAR_OUTPUT
	END_VAR
	VAR_IN_OUT
		machineaxis : FB_AxisCtrl;
	END_VAR
	VAR
		rtrig : R_TRIG;
		timer_tof : TOF;
		merker : BOOL;
		time1_real : REAL;
		time2_real : REAL;
		time_tof : TIME;
		time2 : TP;
		time1 : TP;
		pulse : USINT := 1;
		F_TRIG_2 : F_TRIG;
		F_TRIG_1 : F_TRIG;
		R_TRIG_0 : R_TRIG;
	END_VAR
END_FUNCTION_BLOCK

FUNCTION_BLOCK FB_Liftcrtl (*TODO: Bitte Kommentar hier einfügen*) (*$GROUP=Anwender*)
	VAR_INPUT
		buttomToggle : FB_KeyLamp;
		buttomToggle2 : FB_KeyLamp;
		limiterSwitchDrvSide : BOOL;
		limiterSwitchOpSide : BOOL;
		isup : BOOL;
		isdown : BOOL;
		enable : BOOL;
		init : BOOL;
		onewayini : BOOL;
	END_VAR
	VAR_OUTPUT
		toUp_o : BOOL;
		toDown_o : BOOL;
		limiterBackward_o : BOOL;
		limiterForward_o : BOOL;
	END_VAR
	VAR_IN_OUT
		clk : FB_Clk;
	END_VAR
END_FUNCTION_BLOCK

FUNCTION_BLOCK FB_AxisCtrl_new (*TODO: Bitte Kommentar hier einfügen*) (*$GROUP=Anwender*)
	VAR_INPUT
		Cmd : INT;
		Position : REAL;
		Velocity : REAL;
		Acceleration : REAL;
		Deceleration : REAL;
		Jerk : REAL;
		Override : REAL;
		AxisREF : UDINT;
		BasicControl : basic_typ;
	END_VAR
	VAR_OUTPUT
		busy : BOOL;
		MC_BR_ReadDriveStatus_0 : MC_BR_ReadDriveStatus;
		MC_ReadStatus_0 : MC_ReadStatus;
		err : FB_ErrorHdl;
		MC_ReadActualPosition_0 : MC_ReadActualPosition;
		MC_ReadActualVelocity_0 : MC_ReadActualVelocity;
	END_VAR
	VAR CONSTANT
		STATE_WAIT : USINT := 0; (*NOACTION*)
		STATE_POWER_ON : USINT := 1; (*START*)
		STATE_HOME : USINT := 2; (*CALIBR*)
		STATE_JOG_POSITIVE : USINT := 3;
		STATE_JOG_NEGATIVE : USINT := 4;
		STATE_IDLE : USINT := 5;
		STATE_STOP : USINT := 9;
		STATE_READY : USINT := 10;
		STATE_HALT : USINT := 12;
		STATE_MOVE_ABSOLUTE : USINT := 13;
		STATE_SETPOS : USINT := 14;
		STATE_MOVE_VELOCITY : USINT := 15;
		STATE_MOVE_CYCLIC_VELOCITY : USINT := 20;
		STATE_MOVE_ADDITIVE : USINT := 16;
		STATE_VAXIS_ON : USINT := 17;
		STATE_POWER_OFF : USINT := 18;
		STATE_MOVE_ADDITIVELIMIT : USINT := 19;
		STATE_QUIT : USINT := 98;
		STATE_ERROR_AXIS : USINT := 100;
		STATE_ERROR : USINT := 99;
		STATE_ERROR_RESET : USINT := 102;
	END_VAR
	VAR
		MC_Home_0 : MC_Home;
		MC_BR_CyclicWrite_0 : MC_BR_CyclicWrite;
		CyclicVelocity : REAL;
		MC_MoveAbsolute_0 : MC_MoveAbsolute;
		MC_MoveAdditive_0 : MC_MoveAdditive;
		MC_MoveVelocity_0 : MC_MoveVelocity;
		MC_BR_JogVelocity_0 : MC_BR_JogVelocity;
		MC_BR_JogLimitPosition_0 : MC_BR_JogLimitPosition;
		MC_Power_0 : MC_Power;
		MC_ReadAxisError_0 : MC_ReadAxisError;
		MC_Reset_0 : MC_Reset;
		MC_Stop_0 : MC_Stop;
		MC_Halt_0 : MC_Halt;
		velocityTmp : REAL;
		AxisStep : UINT := STATE_WAIT;
		CONST : FB_CONST_MASCHINE;
		cmdtmp : INT;
		merker : BOOL;
	END_VAR
END_FUNCTION_BLOCK

FUNCTION_BLOCK FB_PACKBELT_DATA (*TODO: Bitte Kommentar hier einfügen*) (*$GROUP=Anwender*)
	VAR_INPUT
		acceleration : REAL;
		deceleration : REAL;
		lowSpeed : REAL;
		highSpeed : REAL;
	END_VAR
END_FUNCTION_BLOCK
```

#### Bibliothek.typ - Lokale Datentypen
```iecst
(********************************************************************
 * COPYRIGHT -- Microsoft
 ********************************************************************
 * Programm: MAIN
 * Datei: MAIN.typ
 * Autor: Awalz
 * Erstellt: 28. März 2014
 ********************************************************************
 * Lokale Datentypen des Programs MAIN
 ********************************************************************)

TYPE
CONST_MACHINE_MODE_Type: STRUCT
	MANUAL:			INT := 0;
	AUTOMATIC:		INT := 1;
	PRODUCTION:		INT := 2;
	SAFETYSTOP:		INT := 7;
	RESET:			INT := 8;
	EMERGENCYSTOP:	INT := 9;
	END_STRUCT;
END_TYPE
```

#### FB_TensionMeasure.st
```iecst
(********************************************************************
 * COPYRIGHT -- Microsoft
 ********************************************************************
 * Library: Bibliothek
 * Datei: FB_TensionMeasure.st
 * Autor: Awalz
 * Erstellt: 12. Mai 2014
 ********************************************************************
 * Implementierung der Library Bibliothek
 ********************************************************************)

 (*<$Description$> TODO: Bitte Kommentar hier einzufügen </$Description$>*)
FUNCTION_BLOCK FB_TensionMeasure
IF init THEN

	LCRPIDpara_TM.Kw						:= 1.0; // No weakening of input
	LCRPIDpara_TM.Kfbk						:= 2.0; // Anti-windup used
	LCRPIDpara_TM.d_mode					:= LCRPID_D_MODE_E;	// differentiate control deviation
	LCRPIDpara_TM.fbk_mode					:= LCRPID_FBK_MODE_INTERN;	// feedback of internal output
	PIDControler.mode						:= LCRPID_MODE_AUTO;	// Standard PID operating mode
	LCRPIDpara_TM.Kp						:= 1.0;
	LCRPIDpara_TM.Tn						:= 0.5;	// Integrative part
	LCRPIDpara_TM.Tv						:= 0.0; // D-part
	LCRPIDpara_TM.Tf						:= 0.020;
	LCRPIDpara_TM.WX_max					:= 1000.0;
	LCRPIDpara_TM.WX_min					:= -1000.0;
	PIDControler.ident						:= LCRPIDpara_TM.ident;
	// Maximum controller output:
	// 50.000 = 3 m/min
	PIDControler.Y_max						:= 100;	// percent
	PIDControler.Y_min						:= -100;	// percent

	// Set output scaling:
	//TensMeas.Data.scaleOut					:= TM_SCALE_PID_OUT_TO_OFFSET;

	//set filter time for tension sensor
	FilterPT1.V	:= 1.0;
	FilterPT1.T1:= TENSION_T_FILTER;
	FilterPT1.enable := TRUE;

	//sign of controller output
	//TensMeas.Para.InverseControl	:= TRUE;// ================
	init := FALSE;
END_IF
	// READ INPUTS
	// ================

		FilterPT1(); (*Eingang filtern*)
		actValue := FilterPT1.y;
			// ================
	// CHECK ERRORS
	// ================

	IF (PIDControler.status > 12022) AND
	   (PIDControler.status < 65534) THEN
		// Error in PID controller detected -> stop control
		(*TensMeas.Data.mainStep		:= STEP_TM_CTRL_OFF;*)

	END_IF

	IF data.mode = CONST.UNITMODEs.DISABLE THEN (* hier noch velocity > 0 detektieren*)
		PIDControler.enable;

	END_IF

	status.mode := data.mode;
	IF status.mode = CONST.UNITMODEs.ENABLE THEN
		status.ready := TRUE;
	ELSE
		status.ready := FALSE;
	END_IF
		PIDControler ();
END_FUNCTION_BLOCK
```

#### Package Logical/Bibliothek/Unwinder - Neues leeres Paket

#### FB_CLAMP.st
```iecst
(********************************************************************
 * COPYRIGHT -- Microsoft
 ********************************************************************
 * Library: Bibliothek
 * Datei: FB_CLAMP_SPLICETABLE.st
 * Autor: Awalz
 * Erstellt: 5. Juni 2014
 ********************************************************************
 * Implementierung der Library Bibliothek
 ********************************************************************)

 (*<$Description$> TODO: Bitte Kommentar hier einzufügen </$Description$>*)
FUNCTION_BLOCK FB_CLAMP
	buttonDown(clk := clk);
	IF disable THEN
		toDown_o := FALSE;
	ELSIF buttonDown.LDT.rtrig.Q (*buttonDown.LDT.button*) THEN
		IF toDown_o THEN
			toDown_o := FALSE;
		ELSE
			toDown_o := TRUE;
		END_IF
	ELSIF visutrigg.Q THEN
		IF toDown_o THEN
			toDown_o := FALSE;
		ELSE
			toDown_o := TRUE;
		END_IF
	END_IF
	buttonDown.LDT.aktion := SEL(toDown_o,CONST.LAMP.OFF, CONST.LAMP.ON);
	visutrigg(CLK := buttonvisu);
END_FUNCTION_BLOCK
```

#### FB_SPLICETABLE.st
```iecst
(********************************************************************
 * COPYRIGHT -- Microsoft
 ********************************************************************
 * Library: Bibliothek
 * Datei: FB_SPLICETABLE.st
 * Autor: Awalz
 * Erstellt: 5. Juni 2014
 ********************************************************************
 * Implementierung der Library Bibliothek
 ********************************************************************)

 (*<$Description$> TODO: Bitte Kommentar hier einzufügen </$Description$>*)
FUNCTION_BLOCK FB_SPLICETABLE
	clampBefore(clk := clk, disable := disable);
	clampAfter(clk := clk, disable := disable);
	ready := NOT clampBefore.toDown_o AND NOT clampAfter.toDown_o;

END_FUNCTION_BLOCK
```

#### FB_Cylinder.st
```iecst
(********************************************************************
 * COPYRIGHT -- Microsoft
 ********************************************************************
 * Library: Bibliothek
 * Datei: FB_Cylinder.st
 * Autor: Awalz
 * Erstellt: 5. Juni 2014
 ********************************************************************
 * Implementierung der Library Bibliothek
 ********************************************************************)

 (*<$Description$> TODO: Bitte Kommentar hier einzufügen </$Description$>*)
FUNCTION_BLOCK FB_Cylinder
	timer(IN := isDown, PT := T#500ms);
	isdowndelayed := timer.Q;
	IF upVISU AND downVISU OR buttonUP AND buttonDown THEN
		;
	ELSIF upVISU OR buttonUP AND NOT isUp THEN
		up_o := TRUE;
		down_o := FALSE;
	ELSIF downVISU OR buttonDown AND NOT isDown THEN
		up_o := FALSE;
		down_o := TRUE;
	ELSE
		up_o := FALSE;
		down_o := FALSE;;
	END_IF
END_FUNCTION_BLOCK
```

#### FB_DUBBLEUUNWINDERDATA.st
```iecst
(********************************************************************
 * COPYRIGHT -- Microsoft
 ********************************************************************
 * Library: Bibliothek
 * Datei: FB_DUBBLEUUNWINDERDATA.st
 * Autor: awalz
 * Erstellt: 24. Juni 2014
 ********************************************************************
 * Implementierung der Library Bibliothek
 ********************************************************************)

(* TODO: Bitte Kommentar hier einfügen *)
FUNCTION_BLOCK FB_DUBBLEUUNWINDERDATA
END_FUNCTION_BLOCK
```

#### FB_UnwinderfeederCtrl.st
```iecst
(********************************************************************
 * COPYRIGHT -- Microsoft
 ********************************************************************
 * Library: Bibliothek
 * Datei: FB_UnwinderfeederCtrl.st
 * Autor: awalz
 * Erstellt: 24. Juni 2014
 ********************************************************************
 * Implementierung der Library Bibliothek
 ********************************************************************)

(* TODO: Bitte Kommentar hier einfügen *)
FUNCTION_BLOCK FB_UnwinderfeederCtrl
		UnwFeeder_HW;
		UnwFeeder_DrvIf;
		UnwFeeder_DiDoIf;

	// INITIALISATION
	IF firststart THEN
	pAxis ACCESS axisREF;
	 (*force variable offset generation *)
	(*pAxis.size                      := pAxis.size;*)

	MC_BR_JogVelocity_0.Axis			:= axisREF;
	MC_BR_JogVelocity_0.Velocity		:= 80.0;
	MC_BR_JogVelocity_0.Acceleration	:= 5000.0;
	MC_BR_JogVelocity_0.Deceleration	:= 5000.0;

	firststart := FALSE;
	END_IF
	buttonLeftOpSide(clk := clk);  			// Taster fahre nach links auf der Antriebsseite
	buttonLeftDrvSide(clk := clk);			// Taster fahre nach links auf der Antriebsseite
	buttonRightOpSide(clk := clk);			// Taster fahre nach rechts auf der Bedienerseite
	buttonRightDrvSide (clk := clk);		// Taster fahre nach rechts auf der Antriebsseite
	buttonRequestOpSide(clk := clk);		// Taster für Rolenwechselanfrage
	buttonRequestDrvSide(clk := clk);		// Taster für Rolenwechselanfrage
	MC_Power_0.Axis := axisREF;
	MC_Stop_0.Axis := axisREF;
	MC_Reset_0.Axis := axisREF;

	(********************MC_BR_READDRIVESTATUS***********************)
	MC_BR_ReadDriveStatus_0.Enable := NOT(MC_BR_ReadDriveStatus_0.Error);
	MC_BR_ReadDriveStatus_0.Axis := axisREF;
	MC_BR_ReadDriveStatus_0.AdrDriveStatus := ADR(BasicControl.Status.DriveStatus);
	(************************ MC_READSTATUS *************************)
	MC_ReadStatus_0.Enable :=  NOT MC_ReadStatus_0.Error;
	MC_ReadStatus_0.Axis := axisREF;
	MC_ReadStatus_0();
//	UnwFeeder_HW. : SdcHwCfg_typ := (0);
//		UnwFeeder_DrvIf.oBrake : SdcDrvIf16_typ := (0);
//		UnwFeeder_DiDoIf : SdcDiDoIf_typ := (0);
	CASE AxisStep OF
	STATE_READY:
			IF cmd <> CONST.AXIS.NOACTION THEN
					busy := TRUE;
					cmdtmp:= cmd;
					IF cmd = CONST.AXIS.RESET THEN
						AxisStep := STATE_ERROR_RESET;
					ELSIF   cmd = CONST.AXIS.POWER_OFF THEN
						AxisStep := STATE_POWER_OFF;
					ELSIF   cmd = CONST.AXIS.POWER_ON THEN
						AxisStep := STATE_POWER_ON;
 					END_IF
			END_IF

	STATE_POWER_ON:
	IF UnwFeeder_ModuleOk AND cmd = CONST.AXIS.POWER_ON AND NOT MC_Power_0.Status
		AND  BasicControl.Status.DriveStatus.ControllerReady AND NOT MC_Power_0.Error  THEN
		MC_Power_0.Enable := TRUE;
	ELSIF	 MC_Power_0.Status THEN
			cmdtmp := cmd;
			AxisStep := STATE_QUIT;
	ELSIF (MC_Power_0.Error AND cmd = CONST.AXIS.POWER_ON ) OR( MC_ReadStatus_0.Errorstop AND cmd = CONST.AXIS.POWER_ON) THEN
			MC_Power_0.Enable := FALSE;
			cmdtmp := cmd;
			cmd := CONST.AXIS.RESET	;
			AxisStep := STATE_ERROR_RESET;
	ELSIF NOT UnwFeeder_ModuleOk OR  NOT BasicControl.Status.DriveStatus.ControllerReady THEN
			cmdtmp := cmd;
			AxisStep := STATE_QUIT;
	END_IF

	STATE_POWER_OFF:
		MC_Power_0.Enable := FALSE;
			IF NOT MC_Power_0.Status THEN
				cmdtmp := cmd;
				(*AxisStep := STATE_READY;*)
				AxisStep := STATE_QUIT;
			END_IF
			(* if a power error occured go to error state *)
			IF MC_Power_0.Error  THEN
				BasicControl.Status.ErrorID := MC_Power_0.ErrorID;
				cmd := CONST.AXIS.RESET;
				AxisStep := STATE_ERROR_RESET;
			END_IF

	STATE_ERROR_RESET:
		IF cmd = CONST.AXIS.RESET THEN
			MC_Power_0.Enable := FALSE;
			MC_Reset_0.Execute := TRUE;
			IF MC_Reset_0.Done THEN
				MC_Reset_0.Execute := FALSE;
				cmdtmp := cmd;
				AxisStep := STATE_QUIT;
			END_IF
		END_IF

	STATE_QUIT:
			busy := FALSE;
			IF cmd = cmdtmp THEN
				busy := FALSE;
				cmd := CONST.AXIS.NOACTION;
				AxisStep := STATE_READY;
			ELSIF cmd <> CONST.AXIS.NOACTION THEN
				busy := FALSE;
				AxisStep := STATE_READY;
			(*ELSIF cmd = CONST.AXIS.POWER_OFF THEN
				cmdtmp := cmd;
				AxisStep := STATE_POWER_OFF;*)
			(*ELSIF cmd = CONST.AXIS.POWER_ON THEN
				cmdtmp := cmd;
				AxisStep := STATE_POWER_ON;*)
			END_IF
	END_CASE

	timer_TP( IN:= Start_timer,PT:= T#1000ms);
	timer_TON(IN := braketimer,PT := T#500ms);
	timerOPside_TOF(IN := buttonRightOpSide.LDT.button OR buttonLeftOpSide.LDT.button OR buttonRequestOpSide.LDT.button,PT := T#40s);
	timerDrvside_TOF(IN := buttonRightDrvSide.LDT.button OR buttonLeftDrvSide.LDT.button OR buttonRequestDrvSide.LDT.button ,PT := T#40s);
	Start_timer := FALSE;
	CASE State OF
	ST_WAIT:
			IF buttonRequestOpSide.LDT.button (*AND  MC_ReadStatus_0.StandStill*) THEN
				brakerelease := FALSE;
				UnwFeeder_DrvIf.oBrake := FALSE;
				horn := TRUE;
				MC_Power_0.Enable := TRUE;
				trigOPSide := TRUE;
				Start_timer := TRUE;
			END_IF

			IF buttonRequestDrvSide.LDT.button (*AND  MC_ReadStatus_0.StandStill*) THEN
				brakerelease := FALSE;
				UnwFeeder_DrvIf.oBrake := FALSE;
				horn := TRUE;
				MC_Power_0.Enable := TRUE;
				Start_timer := TRUE;
				trigDrvSide := TRUE;
//				IF NOT timer_TP.Q THEN
//				State := ST_REQUEST_DrvSide;
//				END_IF
			END_IF
			IF NOT timer_TP.Q AND MC_ReadStatus_0.StandStill AND trigOPSide THEN
				trigOPSide := FALSE;
				State := ST_REQUEST_OpSide;
			ELSIF NOT timer_TP.Q AND MC_ReadStatus_0.StandStill AND trigDrvSide THEN
				trigDrvSide := FALSE;
				State := ST_REQUEST_DrvSide;
			END_IF

		ST_REQUEST_OpSide:
			// Einmal hupen
			// Ampel gelb fängt an zu blinken
			// Taster LED request blinkt
			// beide Abwickler deaktivieren
			// Bremse aus
			MC_BR_JogVelocity_0.Enable	:= TRUE;
			brakerelease := TRUE;
			UnwFeeder_DrvIf.oBrake := TRUE;
			horn := FALSE;
			buttonRequestOpSide.LDT.aktion := CONST.LAMP.ON; (*Zeigt das der Abwickler verfahrbereit ist*)
			IF buttonRequestOpSide.LDT.button AND NOT buttonRightOpSide.LDT.button AND buttonLeftOpSide.LDT.button
				AND LimitSwitchRight THEN
				MC_BR_JogVelocity_0.JogPositive		:= TRUE;
			ELSIF buttonRequestOpSide.LDT.button AND buttonRightOpSide.LDT.button AND NOT buttonLeftOpSide.LDT.button
				 AND LimitSwitchLeft THEN
				MC_BR_JogVelocity_0.JogNegative		:= TRUE;
			ELSE
				MC_BR_JogVelocity_0.JogPositive		:= FALSE;
				MC_BR_JogVelocity_0.JogNegative		:= FALSE;
			END_IF
			IF (buttonRightOpSide.LDT.button AND buttonLeftOpSide.LDT.button) OR NOT timerOPside_TOF.Q THEN
				State := ST_END;
			ELSIF  buttonRequestDrvSide.LDT.button THEN
				MC_BR_JogVelocity_0.JogPositive		:= FALSE;
				MC_BR_JogVelocity_0.JogNegative		:= FALSE;
				State := ST_REQUEST_DrvSide;
			END_IF

		ST_REQUEST_DrvSide:
			MC_BR_JogVelocity_0.Enable	:= TRUE;
			brakerelease := TRUE;
			UnwFeeder_DrvIf.oBrake := TRUE;
			horn := FALSE;
			buttonRequestDrvSide.LDT.aktion := CONST.LAMP.ON; (*Zeigt das der Abwickler verfahrbereit ist*)
			IF buttonRequestDrvSide.LDT.button AND NOT buttonRightDrvSide.LDT.button AND buttonLeftDrvSide.LDT.button
				 AND LimitSwitchLeft THEN
				MC_BR_JogVelocity_0.JogNegative		:= TRUE;
			ELSIF buttonRequestDrvSide.LDT.button AND NOT buttonLeftDrvSide.LDT.button AND buttonRightDrvSide.LDT.button
				AND LimitSwitchRight THEN
				MC_BR_JogVelocity_0.JogPositive		:= TRUE;
			ELSE
				MC_BR_JogVelocity_0.JogPositive		:= FALSE;
				MC_BR_JogVelocity_0.JogNegative		:= FALSE;
			END_IF
			IF (buttonLeftDrvSide.LDT.button AND buttonRightDrvSide.LDT.button) OR NOT timerDrvside_TOF.Q THEN
				State := ST_END;
			ELSIF buttonRequestOpSide.LDT.button THEN
				MC_BR_JogVelocity_0.JogPositive		:= FALSE;
				MC_BR_JogVelocity_0.JogNegative		:= FALSE;
				State := ST_REQUEST_OpSide;
			END_IF

		ST_END:
			MC_BR_JogVelocity_0.Enable	:= FALSE;
			brakerelease := FALSE;
		(*	MC_Power_0.Enable := FALSE;*)
			braketimer := TRUE;
			buttonRequestOpSide.LDT.aktion 	:= CONST.LAMP.OFF;
			buttonRequestDrvSide.LDT.aktion := CONST.LAMP.OFF;
			MC_BR_JogVelocity_0.JogPositive	:= FALSE;
			MC_BR_JogVelocity_0.JogNegative	:= FALSE;
			UnwFeeder_DrvIf.oBrake 			:= FALSE;
			IF timer_TON.Q THEN
				MC_Power_0.Enable := FALSE;
				braketimer := FALSE;
				State := ST_WAIT;
			END_IF
			// Einmal hupen
			// Taster LED blinkt nicht mehr
			// Ampel gelb blinkt nicht mehr
			// beide Abwickler aktivieren
			// Bremse an

	END_CASE
	MC_BR_ReadDriveStatus_0();
	MC_Reset_0();
	MC_Power_0();
	MC_Stop_0();
	MC_BR_JogVelocity_0();

END_FUNCTION_BLOCK
```

#### FB_UNWINDERUNITSTATUS.st
```iecst
(********************************************************************
 * COPYRIGHT -- Microsoft
 ********************************************************************
 * Library: Bibliothek
 * Datei: FB_UNWINDERUNITSTATUS.st
 * Autor: awalz
 * Erstellt: 24. Juni 2014
 ********************************************************************
 * Implementierung der Library Bibliothek
 ********************************************************************)

(* TODO: Bitte Kommentar hier einfügen *)
FUNCTION_BLOCK FB_UNWINDERUNITSTATUS
END_FUNCTION_BLOCK
```

#### Package Logical/Bibliothek/Markpoint_Syncfunc - Paket

#### FB_Markpointarray.st
```iecst
(********************************************************************
 * COPYRIGHT -- Microsoft
 ********************************************************************
 * Library: Bibliothek
 * Datei: FB_Markpointarray.st
 * Autor: awalz
 * Erstellt: 16. Juli 2014
 ********************************************************************
 * Implementierung der Library Bibliothek
 ********************************************************************)

(* TODO: Bitte Kommentar hier einfügen *)
FUNCTION_BLOCK FB_Markpointarray
	bufferRtrig(CLK := new_Ident);
	IF  bufferRtrig.Q THEN (*Arraylist füllen*)
		poslist [ in_posIdent] := rdpos;
		out_posIdent:= in_posIdent - offset_posIdent; (* Berechnung des Offsets für den Druckmarkensensors verschiebung um X Marken zurück*)
		in_posIdent  := in_posIdent + 1;
		// Position Ausgangszeiger vor dem Weitersetzen berechnen
		//		actIdent	:= in_posIdent;

		points[visuIndex].pos := rdpos;
		points[visuIndex].lenght := points[visuIndex].pos - points[visuIndex - 1].pos;
		points[visuIndex].indx := in_posIdent;
		visuIndex := visuIndex + 1;
	END_IF

	maxposIdent := (SIZEOF (poslist) / SIZEOF (poslist[0])) - 1; (* Grpöße der Liste bestimmen*)
	IF in_posIdent > maxposIdent THEN
		in_posIdent := 0;
	END_IF
//		out_posIdent:= in_posIdent - offset_posIdent; (* Berechnung des Offsets für den Druckmarkensensor*)
	IF out_posIdent > maxposIdent THEN
			out_posIdent := out_posIdent + maxposIdent + 1;
	END_IF
//// Abfangen des out_lastIdent INdexes////////////////////////
	out_actIdent := in_posIdent - 1;
	IF out_actIdent > maxposIdent THEN
			out_actIdent := out_actIdent + maxposIdent + 1;
	END_IF
	actpos := poslist [out_actIdent];(* aktulle Markenposition*)
	lastpos:= poslist [ out_posIdent];(*vorletzte bzw Markenposition mit einem Offset von X Markenlängen*)

	IF (in_posIdent > offset_posIdent) AND NOT valid THEN
		valid := TRUE;
	END_IF
	IF reset THEN
		valid := FALSE;
		in_posIdent := 0;
		visuIndex := 0;
		memset(ADR(points), 0, SIZEOF(points));
		reset := FALSE;
	END_IF
	IF visuIndex > maxVisuIndex THEN
		visuIndex := visuIndex - maxVisuIndex - 1;
	END_IF
END_FUNCTION_BLOCK
//
//	VAR_INPUT
//		index :  UDINT;  (**)
//		inpos :  REAL;  (**)
//		new_pos: BOOL
//	END_VAR
//	VAR
//		index :  ARRAY[0..10] OF UDINT;  (**)
//		pos :   ARRAY [0..10] OF REAL;  (**)
//		in_pointer :USINT;
//		out_pointer:USINT;
//		maxpointer: USINT;
//	END_VAR
//	VAR_OUTPUT
//		actpos :REAL;
//		index_out: UDINT;
//	END_VAR
```

#### FB_GetNextCuttPos.st
```iecst
(********************************************************************
 * COPYRIGHT -- Microsoft
 ********************************************************************
 * Library: Bibliothek
 * Datei: FB_GetNextCuttPos.st
 * Autor: awalz
 * Erstellt: 14. Juli 2014
 ********************************************************************
 * Implementierung der Library Bibliothek
 ********************************************************************)

(* TODO: Bitte Kommentar hier einfügen *)
FUNCTION_BLOCK FB_GetNextCuttPos
		(* füllen der Arrayliste*)
		markpoints();
		markpoints.markpointlist();
		setCutOffset.enable := TRUE;  (*Setzen des Korrekturwertes in der Visu*)
		setCutOffset();

		IF markpoints.reset OR reset THEN
			PositionError := 0;
		END_IF
	CASE State OF
		//FIFO is disabled, waiting for Enable
		ST_IDLE:
			PositionErrorValid	:= FALSE;
			PositionError		:= 0;
			indx := 0;
			IF Enable THEN
				State	:= ST_READ_POS;
			END_IF;

		//FIFO is enabled and empty
		ST_READ_POS:
			IF Enable THEN
			(*	IF *)
			(*	masterposMod := REAL_TO_DINT(machinemaster.MC_ReadActualPosition_0.Position);*)
				markposMod :=  (actmarkpos MOD scalePerimeter.ToolSegmentPeriod);
				nextsyncpos := (CutPosition(*(masterposMod - actmarkpos)*) MOD scalePerimeter.ToolSegmentPeriod);(* für die Aufsynchronisierung in Config*)
//				IF ProductLength > 0 THEN
//					markpoints.markpointlist.offset_posIdent := DINT_TO_USINT (DistanceToSensor / ProductLength);
//				END_IF
				IF ProductLength > 0 AND DistanceToSensor < ProductLength THEN
					markpoints.markpointlist.offset_posIdent := DINT_TO_USINT (DistanceToSensor / ProductLength);
				ELSIF DistanceToSensor > ProductLength THEN
					markpoints.markpointlist.offset_posIdent := 0;
				END_IF
				IncompensatinFtrig(CLK := donecut);(*Compensation Ende*)
				IF IncompensatinFtrig.Q THEN
					oldCutPosition := CutPosition;
				END_IF
				IncompensatinRtrig(CLK := donecut);(*Compensation Anfang*)
				IF IncompensatinRtrig.Q THEN
					actCutPosition := CutPosition;
				END_IF
				IF 	IncompensatinRtrig.Q AND newdata <> indx THEN (*CorrectedCutPosition soll nur einmal gespeichert werden und nicht permanent sich ändern*)
				 	 (* wenn TRiggerereignes schon geschenen*)
					tmpCutPosition := actCutPosition;
					newdata := indx;
				ELSIF IncompensatinRtrig.Q AND newdata = indx THEN
					tmpCutPosition := oldCutPosition; (* TRiggerereignes ist nocht nicht geschehen*)
					newdata := indx;
				END_IF
				CorrectedCutPosition	:= markpoints.markpointlist.lastpos + DistanceToSensor +  REAL_TO_DINT (setCutOffset.setOffset_o); (*RegMarkPosition*)
			(*	actmarkpos				:= markpoints.markpointlist.actpos + DistanceToSensor + REAL_TO_DINT (setCutOffset.setOffset_o); (*RegMarkPosition;*)
				IncompensatinRtrig(CLK := donecut);
				IF markpoints.ProbeCounter > 0 AND indx <> markpoints.ProbeCounter (*AND IncompensatinRtrig.Q *) THEN
					indx 				:= markpoints.ProbeCounter;
				END_IF
					IF markpoints.markpointlist.valid THEN (* Wert größer als NULL*)
						(*Position für die Aufsynchronisierung des Querschneiders mit der Annahme das das Messer auf der 0 Position des Zylinders ist*)
						PositionErrorTemp		:=	CorrectedCutPosition  - (*tmpCutPosition;*)CutPosition;
					(*	PositionError			:= markpoints.markpointlist.actpos - markpoints.markpointlist.lastpos - ProductLength;*)(*tatsächliche Abweichung der Marken*)
				(*		newdata := 	indx;*)
						counter := counter + 1;
						IF ABS (PositionErrorTemp) > ProductLength THEN (*Fängt den Überlauf des MC_Touchprobes ab*)
							PositionError := 0;
						ELSE
							IF (PositionErrorTemp < (- ProductLength / 2) ) THEN
								PositionError := PositionErrorTemp + ProductLength;
							ELSIF (PositionErrorTemp > (ProductLength / 2) ) THEN
								PositionError := PositionErrorTemp - ProductLength;
							ELSE
								PositionErrorValid	:= TRUE;
								PositionError := PositionErrorTemp;
							END_IF
						END_IF
						PositionErrorValid	:= FALSE;
					(*	State			:= ST_READ_POS_DONE;*)
					END_IF
			(*	END_IF*)
			ELSE
				State	:= 	ST_IDLE;
			END_IF;

		ST_READ_POS_DONE:
			IF Enable THEN
				IF markpoints.ProbeCounter = indx AND markpoints.ProbeCounter > 0 THEN
					donecounter := donecounter + 1;
				(*	markpoints.new_Ident	:= FALSE;*)
					PositionErrorValid	:= FALSE;
					State	:= ST_READ_POS;
				ELSIF markpoints.ProbeCounter = 0 THEN
					State	:= ST_READ_POS;
				END_IF
			ELSE
				State	:= 	ST_IDLE;
			END_IF
	END_CASE
END_FUNCTION_BLOCK
```

#### FB_Points.st
```iecst
(********************************************************************
 * COPYRIGHT -- Microsoft
 ********************************************************************
 * Library: Bibliothek
 * Datei: FB_Points.st
 * Autor: okrebs
 * Erstellt: 29. Juli 2014
 ********************************************************************
 * Implementierung der Library Bibliothek
 ********************************************************************)

(* TODO: Bitte Kommentar hier einfügen *)
FUNCTION_BLOCK FB_Points
END_FUNCTION_BLOCK
```

#### FB_MarkPoints.st
```iecst
(********************************************************************
 * COPYRIGHT -- Microsoft
 ********************************************************************
 * Library: Bibliothek
 * Datei: FB_MarkPoints.st
 * Autor: awalz
 * Erstellt: 8. Juli 2014
 ********************************************************************
 * Implementierung der Library Bibliothek
 ********************************************************************)

(* TODO: Bitte Kommentar hier einfügen *)
FUNCTION_BLOCK FB_MarkPoints

	IF Enable(* (R_TRIG_Enable.Q)*) THEN
		MC_BR_TouchProbe_0.Axis				:= Axis;
		MC_BR_TouchProbe_0.Period			:= ProductLength;
		MC_BR_TouchProbe_0.PeriodChange		:= 0.0;
		MC_BR_TouchProbe_0.ExpectedValue	:= ProductLength;
		MC_BR_TouchProbe_0.Mode				:= mcSHIFT_FROM_RESULT + mcUSE_FIRST_TRIGGER_POS;
		MC_BR_TouchProbe_0.TriggerInput		:= TriggerInput;
		MC_BR_TouchProbe_0.WindowNegative	:= WindowNegative;
		MC_BR_TouchProbe_0.WindowPositive	:= WindowPositive;
//		GetNextCuttPos.DistanceToSensor		:= DistanceToSensor;
//		GetNextCuttPos.ProductLength		:= REAL_TO_DINT(ProductLength);

	//SearchRM positive edge
	ELSIF Enable AND SearchRM (* R_TRIG_SearchRM.Q*) THEN
		MC_BR_TouchProbe_0.Axis				:= Axis;
		MC_BR_TouchProbe_0.Period			:= ProductLength;
		MC_BR_TouchProbe_0.PeriodChange		:= 0.0;
		MC_BR_TouchProbe_0.ExpectedValue	:= 0.0;
		MC_BR_TouchProbe_0.Mode				:= mcSHIFT_FROM_RESULT + mcUSE_FIRST_TRIGGER_POS;
		MC_BR_TouchProbe_0.TriggerInput		:= TriggerInput;
		MC_BR_TouchProbe_0.WindowNegative	:= WindowNegative;
		MC_BR_TouchProbe_0.WindowPositive	:= WindowPositive;
//		GetNextCuttPos.DistanceToSensor		:= DistanceToSensor;
//		GetNextCuttPos.ProductLength		:= REAL_TO_DINT(ProductLength);
	END_IF

	IF NOT reset THEN
		IF Enable THEN
			MC_BR_TouchProbe_0.Enable	:= TRUE;
		ELSE
			MC_BR_TouchProbe_0.Enable	:= FALSE;
		END_IF
	ELSE
			MC_BR_TouchProbe_0.Enable	:= FALSE;
			ProbeCounter				:= 0;
			MissedTriggers				:= 0;
			reset := FALSE;
			markpointlist.reset := TRUE;
	END_IF
	(* füllen der Arrayliste*)
	MC_BR_TouchProbe_0();

	IF MC_BR_TouchProbe_0.ProbeCounter <> ProbeCounter THEN
		markpointlist.rdpos := MC_BR_TouchProbe_0.RecordedValue;
		lastrecocordedValue := MC_BR_TouchProbe_0.RecordedValue;
		markpointlist.new_Ident := TRUE;
		ProbeCounter := MC_BR_TouchProbe_0.ProbeCounter;
		RecordedValue		:= MC_BR_TouchProbe_0.RecordedValue;
	END_IF
//	markpointlist();
//	markpointlist.new_Ident := FALSE;
	IF MC_BR_TouchProbe_0.MissedTriggers <> MissedTriggers AND MC_BR_TouchProbe_0.ProbeCounter = ProbeCounter THEN (* soweit eine Marke verloren gegangen ist, wird feste Länge jedesmal dazu addiert*)
		markpointlist.rdpos := lastrecocordedValue + REAL_TO_DINT (ProductLength);(*(ActProductLength);*)
	(*	markpointlist.rdpos := MC_BR_TouchProbe_0.RecordedValue;*)
		lastrecocordedValue := markpointlist.rdpos;
		markpointlist.new_Ident := TRUE;
		MissedTriggers := MC_BR_TouchProbe_0.MissedTriggers;
		RecordedValue		:= markpointlist.rdpos;
	END_IF
	markpointlist();
	markpointlist.new_Ident := FALSE;
	//update FUB outputs
//	RecordedValue		:= MC_BR_TouchProbe_0.RecordedValue;
//	ProbeCounter		:= MC_BR_TouchProbe_0.ProbeCounter;
	(*MissedTriggers		:= MC_BR_TouchProbe_0.MissedTriggers;*)
	Busy				:= Enable OR MC_BR_TouchProbe_0.Busy;
	Active				:= MC_BR_TouchProbe_0.Active;

	IF MC_BR_TouchProbe_0.Active THEN
		ActProductLength	:= MC_BR_TouchProbe_0.Period + MC_BR_TouchProbe_0.DeltaExpectedValue;
	ELSE
		ActProductLength	:= 0.0;
	END_IF;

	IF MC_BR_TouchProbe_0.Enable THEN
		Error	:= MC_BR_TouchProbe_0.Error;
		ErrorID	:= MC_BR_TouchProbe_0.ErrorID;
	ELSIF NOT Enable THEN
		Error	:= FALSE;
		ErrorID	:= FALSE;
	END_IF;
END_FUNCTION_BLOCK
```

#### FB_SafeInputs.st
```iecst
(********************************************************************
 * COPYRIGHT -- Microsoft
 ********************************************************************
 * Library: Bibliothek
 * Datei: FB_SafeInputs.st
 * Autor: awalz
 * Erstellt: 15. Juli 2014
 ********************************************************************
 * Implementierung der Library Bibliothek
 ********************************************************************)

(* TODO: Bitte Kommentar hier einfügen *)
FUNCTION_BLOCK FB_SafeInputs

		EMCY_Button1_o.0 	:= EMCY_Button1;
		EMCY_Button2_o.0 	:= EMCY_Button2;
		EMCY_Button3_o.0 	:= EMCY_Button3;
		EMCY_Button4_o.0 	:= EMCY_Button4;
		EMCY_Door1_o.0 		:= EMCY_Door1;
		EMCY_Door2_o.0 		:= EMCY_Door2;
		EMCY_Door3_o.0 		:= EMCY_Door3;
		EMCY_Door4_o.0 		:= EMCY_Door4;
		EMCY_Door5_o.0 		:= EMCY_Door5;
		EMCY_Door6_o.0 		:= EMCY_Door6;
		EMCY_pullwireOPs_o.0:=EMCY_pullwireOPs;
		EMCY_pullwireDVRs_o.0:=EMCY_pullwireDVRs;
END_FUNCTION_BLOCK
```

#### FB_HandWheel.st
```iecst
(********************************************************************
 * COPYRIGHT -- Microsoft
 ********************************************************************
 * Library: Bibliothek
 * Datei: FB_HandWheel.st
 * Autor: okrebs
 * Erstellt: 31. Juli 2014
 ********************************************************************
 * Implementierung der Library Bibliothek
 ********************************************************************)

(* TODO: Bitte Kommentar hier einfügen *)
FUNCTION_BLOCK FB_HandWheel
	IF safetyspeedrequest THEN	(* Safetyspeed ist quttiert Maschine kann schneller als 4.9m/min fahren*)
		IF (lastCounterValue < counterHandWheel) THEN
			setVelocity := (actualVelocity + velocityStep)/16666.67;
		ELSIF (lastCounterValue > counterHandWheel) THEN
			setVelocity := (actualVelocity - velocityStep)/16666.67;
		END_IF;
		setVelocity := LIMIT (1, setVelocity, limitspeed/16666.67);
		lastCounterValue := counterHandWheel;
		IF reset THEN
			setVelocity := 1;
			(*actualVelocity := 0;*)
			reset := FALSE;
		END_IF
	ELSE (* falls die Safetyspeed nicht quttiert war Geschwindkeit auf 3.9m/min begrenzen 3.9*16666,67=65000.67**)
		IF (lastCounterValue < counterHandWheel) THEN
			setVelocity := (actualVelocity + velocityStep)/16666.67;
		ELSIF (lastCounterValue > counterHandWheel) THEN
			setVelocity := (actualVelocity - velocityStep)/16666.67;
		END_IF;
		setVelocity := LIMIT (1, setVelocity,65000/16666.67); (*weil man davor so bescheident war und ständig umgerechnet hat muss es auch hier passieren*)
		lastCounterValue := counterHandWheel;
		IF reset THEN
			setVelocity := 1;
			(*actualVelocity := 0;*)
			reset := FALSE;
		END_IF
	END_IF
END_FUNCTION_BLOCK
```

### Package Logical/MainMachineCtrl - General Machine Functions and Master axis

### Program Logical/MainMachineCtrl/ncsdcctrl (IEC)

#### ncsdcctrl.st
```iecst
PROGRAM _INIT

	(* initialize variables *)
	gUnwFeeder_HW.DrvIf_Typ := ncSDC_DRVSERVO16;
	strcpy( ADR(gUnwFeeder_HW.DrvIf_Name[0]), ADR('gUnwFeeder_DrvIf') );
	gUnwFeeder_HW.DiDoIf_Typ := ncSDC_DIDO;
	strcpy( ADR(gUnwFeeder_HW.DiDoIf_Name[0]), ADR('gUnwFeeder_DiDoIf') );

	(* force variable offset generation *)
	gUnwFeeder.size                      := gUnwFeeder.size;
	gUnwFeeder_DrvIf.iLifeCnt            := gUnwFeeder_DrvIf.iLifeCnt;
	gUnwFeeder_DiDoIf.iLifeCntDriveReady := gUnwFeeder_DiDoIf.iLifeCntDriveReady;
	gUnwFeeder_ModuleOk                  := gUnwFeeder_ModuleOk;

(* ### BEGIN gPackBelt ### *)

(* initialize variables *)
 gPackBelt_HW.DrvIf_Typ := ncSDC_DRVSERVO16;
 strcpy( ADR(gPackBelt_HW.DrvIf_Name[0]), ADR('gPackBelt_DrvIf') );
 gPackBelt_HW.DiDoIf_Typ := ncSDC_DIDO;
 strcpy( ADR(gPackBelt_HW.DiDoIf_Name[0]), ADR('gPackBelt_DiDoIf') );

(* force variable offset generation *)
 gPackBelt.size                      := gPackBelt.size;
 gPackBelt_DrvIf.iLifeCnt            := gPackBelt_DrvIf.iLifeCnt;
 gPackBelt_DiDoIf.iLifeCntDriveReady := gPackBelt_DiDoIf.iLifeCntDriveReady;
 gPackBelt_ModuleOk                  := gPackBelt_ModuleOk;

(* assign your hardware inputs here*)

(* gPackBelt_DiDoIf.iPosHwEnd  := gPackBelt_DiDoIf.iPosHwEnd;
 gPackBelt_DiDoIf.iNegHwEnd  := gPackBelt_DiDoIf.iNegHwEnd;
 gPackBelt_DiDoIf.iReference := gPackBelt_DiDoIf.iReference;
 *)

(* ### END gPackBelt ### *)

END_PROGRAM

PROGRAM _CYCLIC

(* ### BEGIN gLaminator ### *)
(* life counter emulation of digital inputs *)
	gUnwFeeder_DiDoIf.iLifeCntReference := gUnwFeeder_DiDoIf.iLifeCntReference + 1;
	gUnwFeeder_DiDoIf.iLifeCntNegHwEnd  := gUnwFeeder_DiDoIf.iLifeCntNegHwEnd  + 1;
	gUnwFeeder_DiDoIf.iLifeCntPosHwEnd  := gUnwFeeder_DiDoIf.iLifeCntPosHwEnd  + 1;
(* ### END gLaminator ### *)

(* ### BEGIN gPackBelt ### *)

(* life counter emulation of digital inputs *)
 gPackBelt_DiDoIf.iLifeCntReference := gPackBelt_DiDoIf.iLifeCntReference + 1;
 gPackBelt_DiDoIf.iLifeCntNegHwEnd  := gPackBelt_DiDoIf.iLifeCntNegHwEnd  + 1;
 gPackBelt_DiDoIf.iLifeCntPosHwEnd  := gPackBelt_DiDoIf.iLifeCntPosHwEnd  + 1;

	(* ### END gPackBelt ### *)

END_PROGRAM
```

### Program Logical/MainMachineCtrl/MAIN (IEC) - Ein neues Programm

#### MAIN.st - Zyklischer Code
```iecst
(********************************************************************
 * COPYRIGHT -- Microsoft
 ********************************************************************
 * Programm: MAIN
 * Datei: MAIN.st
 * Autor: Awalz
 * Erstellt: 25. März 2014
 ********************************************************************
 * Implementierung des Programms MAIN
 ********************************************************************)
PROGRAM _INIT
	gNewOutputBrake;
	(* Zuweisung der Achsvar*)
	machine.masterModul.axis.AxisREF:= ADR(gMaster1);
	machine.UnwinderUnit.unwinderDrv.unwinderaxis.AxisREF := ADR (gUnwDrv);
	machine.UnwinderUnit.unwinderOp.unwinderaxis.AxisREF := ADR (gUnwOp);

	machine.webbuffer.axis.ctrl.AxisREF := ADR(gBuffer);
	machine.webbuffer.axis.bufferaxis.AxisREF := ADR(gBuffer);
	machine.webbuffer.axis.refSwitchConfig.Axis := ADR(gBuffer);

	machine.pullbreak.axis.ctrl.AxisREF:= ADR (gPBS1);
	machine.pullbreakSt.axis.ctrl.AxisREF := ADR (gPBS2);
	machine.UnwinderUnit.feederCtrl.axisREF := ADR(gUnwFeeder);
	// neu // OKrebs // 23.11.16
	machine.packbelt.ctrl.axisREF := ADR(gPackBelt);
	// ende neu
	machine.cuttingunit1.axis.ctrl.AxisREF := ADR(gCut1);
	machine.cuttingunit1.axis.refSwitchConfig.Axis := ADR(gCut1);

//	machine.cuttingunit1.markpoints.TriggerInput.Edge			:= ncP_EDGE;
//	machine.cuttingunit1.markpoints.TriggerInput.EventSourceParID:= ACP10PAR_STAT_TRIGGER1;
//	machine.cuttingunit1.markpoints.TriggerInput.MaxWidth		:= 0;
//	machine.cuttingunit1.markpoints.TriggerInput.MinWidth		:= 0;
//	machine.cuttingunit1.markpoints.TriggerInput.ProbeParID		:= ACP10PAR_MA1_CYCLIC_POS;
//	machine.cuttingunit1.markpoints.TriggerInput.SensorDelay	:= -25;

	machine.turngridwinder.gridwinderleft.axis.AxisREF := ADR(gGridLeft);
	machine.turngridwinder.gridwinderright.axis.AxisREF := ADR(gGridRight);
	machine.turngridwinder.feeder.AxisREF := ADR(gGridFeeder);
	// neu // OKrebs // 13.04.17
	machine.turngridwinder.ctrl.refSwitchConfig.Axis := ADR(gGridFeeder);
	machine.turngridwinder.ctrl.SwitchConfig.Axis := ADR(gGridFeeder);
	// ende neu
	machine.longcutter.axis.ctrl.AxisREF := ADR(gLongCut);

	machine.cuttingunit2.axis.ctrl.AxisREF := ADR (gCut2);
	machine.cuttingunit2.axis.refSwitchConfig.Axis := ADR (gCut2);

	machine.cuttingunit2.markpoints.TriggerInput.Edge			:= ncP_EDGE;
	machine.cuttingunit2.markpoints.TriggerInput.EventSourceParID:= ACP10PAR_STAT_TRIGGER1;
	machine.cuttingunit2.markpoints.TriggerInput.MaxWidth		:= 0;
	machine.cuttingunit2.markpoints.TriggerInput.MinWidth		:= 0;
	machine.cuttingunit2.markpoints.TriggerInput.ProbeParID		:= ACP10PAR_MA1_CYCLIC_POS;
	machine.cuttingunit2.markpoints.TriggerInput.SensorDelay	:= -900;

	machine.catchbelt.axis.ctrl.AxisREF := ADR(gCatchBelt);

	machine.conveyor.axis.ctrl.AxisREF := ADR (gConvBelt);
	machine.gVarMachine.gMachine := gMachine;

	machine.UnwinderUnit.unwinderOp.data.machData.GEAR_RATIO := 8;

	machine.UnwinderUnit.unwinderDrv.data.machData.GEAR_RATIO := 8;

	machine.turngridwinder.gridwinderleft.data.machData.GEAR_RATIO := 3;

	machine.turngridwinder.gridwinderright.data.machData.GEAR_RATIO := 3;

	machine.webbuffer.data.machData.GEAR_RATIO := 12;

	LayerStatus						:= 1;

	machine.cuttingunit2.data.recipe.MaxCorr := 200000;

	// Beim Einschalten wird das aktuelle Rezept und Maschinendaten in die MAIN-Bausteinvariablen geladen //////
	ac_loadRecipeMain;
	ac_saveMachData;
	//////////////////////////////////////////////////////////////////////////////////////////////////////////////////////////

	machine.cuttingunit1.data.recipe.tool.gearRatioMotor := 5;
	machine.cuttingunit1.data.recipe.tool.cogmodul :=3175.0;
	machine.cuttingunit2.data.recipe.tool.gearRatioMotor := 5;
	machine.cuttingunit2.data.recipe.tool.cogmodul :=3175.0;
END_PROGRAM

PROGRAM _CYCLIC
(*machine.cuttingunit1.axis.ctrl.ACP10AXIS := gCut1;*)
//machine.IOs.aIn := gMachine.IO.AIn;
//machine.IOs.aOut := gMachine.IO.AOut;
//machine.IOs.dIn := gMachine.IO.DIn;
//machine.IOs.dOut := gMachine.IO.DOut;
//machine.cuttingunit1.data.recipe := gApplRecipe.cutUnit1; (*Rezepte sind noch nicht bereit*)
	machine.UnwinderUnit.feederCtrl.UnwFeeder_DiDoIf := gUnwFeeder_DiDoIf;
	machine.UnwinderUnit.feederCtrl.UnwFeeder_DrvIf := gUnwFeeder_DrvIf;
// 24.7.2024 - Change braking DO logic ---	gUnwFeeder_DrvIf.oBrake := machine.UnwinderUnit.feederCtrl.UnwFeeder_DrvIf.oBrake;
	machine.UnwinderUnit.feederCtrl.UnwFeeder_HW  := gUnwFeeder_HW;
	machine.UnwinderUnit.feederCtrl.UnwFeeder_ModuleOk := gUnwFeeder_ModuleOk;

	/// neu // OKrebs // 23.11.16
	machine.packbelt.ctrl.PackBelt_DiDoIf := gPackBelt_DiDoIf;
	machine.packbelt.ctrl.PackBelt_DrvIf := gPackBelt_DrvIf;
	machine.packbelt.ctrl.PackBelt_HW := gPackBelt_HW;
	machine.packbelt.ctrl.PackBelt_ModuleOk := gPackBelt_ModuleOk;
// 24.7.2024 - Change braking DO logic ---	gUnwFeeder_DrvIf.oBrake := machine.packbelt.ctrl.PackBelt_DrvIf.oBrake;
	// ende neu

	// 24.7.2024 - Change braking DO logic
	IF machine.packbelt.ctrl.PackBelt_DrvIf.oBrake OR machine.UnwinderUnit.feederCtrl.UnwFeeder_DrvIf.oBrake THEN
		gUnwFeeder_DrvIf.oBrake := TRUE;
		LocalNewOutputBrake := TRUE;
		gNewOutputBrake := TRUE;

	ELSIF  machine.packbelt.ctrl.PackBelt_DrvIf.oBrake = 0 AND machine.UnwinderUnit.feederCtrl.UnwFeeder_DrvIf.oBrake = 0 THEN
		gUnwFeeder_DrvIf.oBrake := FALSE;
		LocalNewOutputBrake := FALSE;
		gNewOutputBrake := FALSE;
	END_IF;

	// neu // OKrebs // 26.04.17
	TOF_OutputGrinderON(IN := machine.masterModul.axis.MC_ReadStatus_0.ContinuousMotion, PT := T#60s);
	OutputGrinderON := TOF_OutputGrinderON.Q;
	// ende neu
	// neu // OKrebs // 27.04.17
	machine.conveyor.counters.manualButton := machine.packbelt.ctrl.buttonStart;
	// neu ende
	//	machine.cuttingunit1.data.machdata := gMachRecipe.cut1;
	//
	//	machine.cuttingunit1.data.recipe.mode := 1 ;
	//	machine.cuttingunit1.data.recipe.markPointNo := 1;
	//	machine.cuttingunit1.data.recipe.MaxCorr := 300000;
	//	machine.cuttingunit1.data.recipe.tool.numberToolSegments := 1;
	//	machine.cuttingunit1.data.recipe.toolNumber :=1;
	//	machine.cuttingunit1.data.recipe.tool.cogCutting := 145;(*Werkzeug*)
	//	machine.cuttingunit1.data.recipe.tool.cogSupportSpindle := 160;(*Stützwelle*)
	//	machine.cuttingunit1.data.recipe.tool.cutEndPosition := 300000; (*Umfang = 460,375*)
	//	machine.cuttingunit1.data.recipe.tool.cutStartPosition := 0;
	//	machine.cuttingunit1.data.general.periodLength := 460000; (* 460000 *)
	//	machine.cuttingunit1.data.general.startVelocity := 10000;
	//	machine.cuttingunit1.data.general.maxVelocity := 40000;
	//	machine.cuttingunit1.data.general.masterAcceleration := 60000;
	//	machine.cuttingunit1.data.general.masterDeceleration := 60000;

	//machine.cuttingunit2.data.recipe := gApplRecipe.cutUnit2;
	//machine.cuttingunit2.data.machdata := gMachRecipe.cut2;
	//
	//	machine.cuttingunit2.data.recipe.mode := 3;
	//	//machine.cuttingunit2.data.recipe.MaxCorr := 30000;
	//	machine.cuttingunit2.data.recipe.tool.numberToolSegments := 1;
	//	machine.cuttingunit2.data.recipe.toolNumber :=1;
	//	machine.cuttingunit2.data.recipe.tool.cogCutting := 189;(*Werkzeug*)
	//	machine.cuttingunit2.data.recipe.tool.cogSupportSpindle := 160;(*Stützwelle*)
	//	machine.cuttingunit2.data.recipe.tool.cutEndPosition := 550000; (*Umfang = 460,375*)
	//	machine.cuttingunit2.data.recipe.tool.cutStartPosition := 50000;(*20000*)
	//
	//	machine.cuttingunit2.data.general.periodLength := 430000; (*410000; TEst*)
	//	machine.cuttingunit2.data.recipe.RmWindow := 30000;
	//	machine.cuttingunit2.data.machdata.position := 540000;

	///////////////////  Rezept aktivieren ////////////////////////////////////////////////////////////////////////////////////
	IF gMachine.Command.UpdateRecipe AND (machine.ctrl.mode.ctrl.value = CONST.MACHINEMODES.MANUAL OR machine.ctrl.mode.ctrl.value = CONST.MACHINEMODES.EMERGENCYSTOP) THEN
		gMachine.Command.UpdateRecipe := FALSE;
		ac_loadRecipeMain;
	END_IF
	///////////////////////////////////////////////////////////////////////////////////////////////////////////////////////

	/////////////  Kopieren der Rezeptdaten aus MAIN zu RecipeEdit (Laden aus Maschine Button) ////////////////////////////
	IF Button.F3 = 1 AND machine.ctrl.mode.ctrl.value = CONST.MACHINEMODES.MANUAL THEN
		Button.F3 := 0;
		ac_loadMach_toRecipeMain;
	END_IF
	//////////////////////////////////////////////////////////////////////////////////////////////////////////////////////

	///////////// Speichern der Maschienendaten von gMachData zu MAIN-Variablen	///////////////////////////////////////////
	IF SaveMachData AND (machine.ctrl.mode.ctrl.value = CONST.MACHINEMODES.MANUAL OR machine.ctrl.mode.ctrl.value = CONST.MACHINEMODES.EMERGENCYSTOP) THEN
		SaveMachData := FALSE;
		ac_saveMachData;
	END_IF
	///////////////////////////////////////////////////////////////////////////////////////////////////////////////////////

	machine.cuttingunit2.markpoints();
	machine(); (* Aufruf der Machine bzw. des FB_Machine*)
	//////////////////////////////////////////////////////////////////////////////////////////////////////////////////////

	IF machine.UnwinderUnit.unwinderDrv.data.recipeData.mode = 1 THEN
		machine.IOs.Unwinder_Drv_Led := TRUE;
	ELSE
		machine.IOs.Unwinder_Drv_Led := FALSE;
	END_IF

	IF machine.UnwinderUnit.unwinderOp.data.recipeData.mode = 1 THEN
		machine.IOs.Unwinder_OP_Led := TRUE;
	ELSE
		machine.IOs.Unwinder_OP_Led := FALSE;
	END_IF

	UnwinderOPModeTrig(CLK :=machine.IOs.Unwinder_OP_Button );

	IF UnwinderOPModeTrig.Q = TRUE AND machine.UnwinderUnit.unwinderOp.data.recipeData.mode = 2 THEN
		machine.UnwinderUnit.unwinderOp.data.recipeData.mode := 1;
	ELSE
		IF UnwinderOPModeTrig.Q = TRUE AND machine.UnwinderUnit.unwinderOp.data.recipeData.mode = 1 THEN
			machine.UnwinderUnit.unwinderOp.data.recipeData.mode :=2;
		ELSE
		END_IF
	END_IF

	UnwinderDRVModeTrig(CLK:=machine.IOs.Unwinder_Drv_Button );

	IF UnwinderDRVModeTrig.Q = TRUE AND machine.UnwinderUnit.unwinderDrv.data.recipeData.mode = 2 THEN
		machine.UnwinderUnit.unwinderDrv.data.recipeData.mode := 1;
	ELSE
		IF UnwinderDRVModeTrig.Q = TRUE AND machine.UnwinderUnit.unwinderDrv.data.recipeData.mode = 1 THEN
			machine.UnwinderUnit.unwinderDrv.data.recipeData.mode :=2;
		ELSE
		END_IF
	END_IF
	machine.IOs.aIn.Dancer_position.Config.ScaleGain := 0.03357;
	machine.IOs.aIn.Dancer_position.Config.ScaleOffset := 200;
	machine.IOs.aIn.Dancer_position.Value.Scaled := machine.IOs.aIn.Dancer_position.Value.RawInt*machine.IOs.aIn.Dancer_position.Config.ScaleGain-machine.IOs.aIn.Dancer_position.Config.ScaleOffset;

	IF EDGENEG(gMachine.IO.DIn.Liner_detekce.Value.State)AND machine.masterModul.axis.MC_ReadActualVelocity_0.Velocity > 0.0 THEN
		machine.ctrl.alarms.alarmlist[49] := TRUE;
	END_IF

	IF gMachine.IO.DIn.LDT_FaultReset.Value.InVal OR machine.masterModul.axis.MC_ReadActualVelocity_0.Velocity = 0.0 THEN
		machine.ctrl.alarms.alarmlist[49] := FALSE;
	END_IF

END_PROGRAM
```

#### MAIN.var - Lokale Variablen
```iecst
(********************************************************************
 * COPYRIGHT -- Microsoft
 ********************************************************************
 * Programm: MAIN
 * Datei: MAIN.var
 * Autor: Awalz
 * Erstellt: 25. März 2014
 ********************************************************************
 * Lokale Variablen des Programms MAIN
 ********************************************************************)
(*CONST : 	CONST_MACHINE_MODES:= (0);*)
(*CONST : CONST_MACHINE_MODES_Type:=(MANUAL:=0,AUTOMATIC:=1,PRODUCTION:=2,SAFETYSTOP:=7,RESET:=8,EMERGENCYSTOP:=9);*)
(*CONST : CONST_MACHINE_MODES_Type := MANUAL;*)
VAR CONSTANT
	ST_IDLE : INT := 0;
	ST_SAFETYSTOP : INT := 1;
	ST_MANUAL : INT := 2;
	ST_AUTO : INT := 3;
	ST_PRODUCTION : INT := 4;
	SCALE_MM_TO_DRIVE_UNITS : REAL := 1000.0; (*mm to micrometer (drive units)*)
END_VAR
VAR
	machine : FB_Machine;
	LayerStatus : INT := 0; (*refSwitchDevNameCut1 : STRING[80]; (*Device name for reference switch input (X20)*) (*refSwitchChNameCut1 : STRING[80];*)
	SaveMachData : BOOL;
	CONST : FB_CONST_MASCHINE;
	R_TRIG_0 : R_TRIG;
	UnwinderOPModeTrig : R_TRIG;
	UnwinderDRVModeTrig : R_TRIG;
	OutputGrinderON : BOOL;
	TOF_OutputGrinderON : TOF;
	endif : BOOL;
	NewoBrake : BOOL;
	LocalNewOutputBrake : BOOL;
END_VAR
```
